C03644=1019.248,-10.777,397.334,166.343,52.857,159.580
C03645=1019.242,-11.026,397.348,166.340,52.863,159.581
C03646=1019.236,-11.276,397.360,166.337,52.868,159.581
C03647=1019.231,-11.525,397.374,166.334,52.874,159.582
C03648=1019.225,-11.775,397.386,166.331,52.880,159.582
C03649=1019.220,-12.024,397.400,166.328,52.885,159.583
C03650=1019.214,-12.274,397.413,166.325,52.891,159.583
C03651=1019.208,-12.523,397.426,166.322,52.896,159.583
C03652=1019.203,-12.773,397.439,166.321,52.902,159.584
C03653=1019.197,-13.023,397.451,166.318,52.907,159.584
C03654=1019.192,-13.272,397.465,166.315,52.913,159.585
C03655=1019.186,-13.522,397.478,166.312,52.919,159.586
C03656=1019.180,-13.771,397.490,166.309,52.924,159.586
C03657=1019.175,-14.021,397.504,166.306,52.929,159.586
C03658=1019.169,-14.271,397.516,166.303,52.935,159.587
C03659=1019.164,-14.521,397.530,166.301,52.941,159.587
C03660=1019.158,-14.770,397.542,166.299,52.946,159.588
C03661=1019.153,-15.020,397.555,166.296,52.951,159.588
C03662=1019.147,-15.269,397.569,166.293,52.957,159.589
C03663=1019.141,-15.519,397.581,166.290,52.962,159.589
C03664=1019.137,-15.769,397.594,166.287,52.968,159.590
C03665=1019.130,-16.018,397.607,166.284,52.974,159.590
C03666=1019.124,-16.268,397.620,166.281,52.979,159.591
C03667=1019.118,-16.518,397.632,166.279,52.985,159.591
C03668=1019.113,-16.767,397.645,166.276,52.991,159.592
C03669=1019.108,-17.016,397.658,166.273,52.996,159.592
C03670=1019.102,-17.266,397.671,166.270,53.002,159.593
C03671=1019.096,-17.515,397.683,166.267,53.007,159.593
C03672=1019.091,-17.765,397.696,166.265,53.014,159.594
C03673=1019.085,-18.015,397.708,166.263,53.019,159.594
C03674=1019.079,-18.265,397.721,166.260,53.024,159.595
C03675=1019.073,-18.514,397.733,166.257,53.030,159.595
C03676=1019.068,-18.764,397.747,166.254,53.035,159.596
C03677=1019.062,-19.014,397.759,166.251,53.041,159.596
C03678=1019.057,-19.263,397.772,166.249,53.047,159.597
C03679=1019.051,-19.513,397.784,166.246,53.052,159.597
C03680=1019.045,-19.763,397.797,166.243,53.058,159.597
C03681=1019.040,-20.012,397.809,166.240,53.064,159.598
C03682=1019.034,-20.262,397.821,166.237,53.069,159.598
C03683=1019.028,-20.512,397.834,166.234,53.075,159.599
C03684=1019.023,-20.761,397.847,166.231,53.080,159.599
C03685=1019.016,-21.039,397.861,166.229,53.086,159.600
C03686=1019.010,-21.317,397.875,166.225,53.093,159.600
C03687=1019.004,-21.596,397.888,166.223,53.099,159.601
C03688=1018.998,-21.874,397.903,166.219,53.105,159.601
C03689=1018.992,-22.124,397.915,166.216,53.111,159.602
C03690=1018.986,-22.374,397.928,166.213,53.117,159.602
C03691=1018.981,-22.623,397.940,166.210,53.122,159.603
C03692=1018.975,-22.873,397.952,166.207,53.128,159.603
C03693=1018.970,-23.122,397.965,166.204,53.133,159.604
C03694=1018.964,-23.372,397.978,166.201,53.139,159.604
C03695=1018.958,-23.622,397.991,166.199,53.145,159.605
C03696=1018.953,-23.872,398.002,166.197,53.150,159.605
C03697=1018.947,-24.122,398.015,166.194,53.155,159.605
C03698=1018.942,-24.371,398.027,166.191,53.161,159.606
C03699=1018.936,-24.621,398.040,166.189,53.167,159.607
C03700=1018.931,-24.870,398.052,166.186,53.172,159.607
C03701=1018.925,-25.120,398.064,166.183,53.177,159.607
C03702=1018.919,-25.370,398.077,166.180,53.183,159.608
C03703=1018.914,-25.619,398.090,166.177,53.188,159.608
C03704=1018.909,-25.869,398.102,166.174,53.194,159.609
C03705=1018.903,-26.118,398.115,166.171,53.200,159.609
C03706=1018.897,-26.368,398.127,166.168,53.205,159.609
C03707=1018.892,-26.617,398.139,166.165,53.211,159.610
C03708=1018.886,-26.867,398.152,166.163,53.216,159.610
C03709=1018.881,-27.116,398.164,166.160,53.221,159.611
C03710=1018.875,-27.366,398.177,166.157,53.227,159.611
C03711=1018.870,-27.616,398.188,166.155,53.233,159.612
C03712=1018.864,-27.866,398.201,166.152,53.238,159.612
C03713=1018.858,-28.116,398.213,166.149,53.244,159.613
C03714=1018.853,-28.365,398.225,166.146,53.250,159.613
C03715=1018.847,-28.615,398.237,166.143,53.255,159.614
C03716=1018.842,-28.865,398.249,166.140,53.261,159.614
C03717=1018.835,-29.114,398.261,166.137,53.266,159.614
C03718=1018.830,-29.363,398.274,166.135,53.272,159.615
C03719=1018.825,-29.613,398.285,166.132,53.278,159.615
C03720=1018.819,-29.863,398.298,166.129,53.283,159.616
C03721=1018.814,-30.112,398.310,166.126,53.289,159.616
C03722=1018.808,-30.363,398.322,166.123,53.295,159.617
C03723=1018.802,-30.612,398.333,166.120,53.300,159.617
C03724=1018.796,-30.862,398.346,166.118,53.306,159.618
C03725=1018.791,-31.111,398.357,166.115,53.312,159.618
C03726=1018.785,-31.361,398.370,166.112,53.317,159.619
C03727=1018.780,-31.610,398.382,166.109,53.322,159.619
C03728=1018.774,-31.861,398.394,166.107,53.329,159.620
C03729=1018.768,-32.110,398.405,166.104,53.334,159.620
C03730=1018.763,-32.359,398.418,166.101,53.339,159.620
C03731=1018.757,-32.609,398.429,166.098,53.345,159.621
C03732=1018.752,-32.859,398.442,166.095,53.350,159.621
C03733=1018.746,-33.109,398.454,166.092,53.356,159.622
C03734=1018.740,-33.358,398.465,166.089,53.362,159.622
C03735=1018.734,-33.608,398.478,166.086,53.367,159.623
C03736=1018.729,-33.858,398.489,166.083,53.373,159.623
C03737=1018.724,-34.107,398.501,166.081,53.379,159.624
C03738=1018.718,-34.357,398.514,166.078,53.384,159.624
C03739=1018.713,-34.606,398.525,166.075,53.390,159.624
C03740=1018.707,-34.855,398.537,166.072,53.395,159.625
C03741=1018.702,-35.106,398.549,166.069,53.401,159.625
C03742=1018.696,-35.355,398.561,166.066,53.406,159.626
C03743=1018.691,-35.606,398.573,166.064,53.412,159.626
C03744=1018.685,-35.855,398.585,166.061,53.418,159.627
C03745=1018.680,-36.104,398.596,166.058,53.423,159.627
C03746=1018.674,-36.354,398.608,166.055,53.429,159.627
C03747=1018.669,-36.604,398.620,166.052,53.434,159.628
C03748=1018.663,-36.853,398.632,166.049,53.440,159.628
C03749=1018.658,-37.081,398.642,166.047,53.445,159.629
C03750=1018.653,-37.308,398.654,166.044,53.450,159.629
C03751=1018.649,-37.536,398.664,166.040,53.455,159.629
C03752=1018.643,-37.764,398.674,166.039,53.460,159.630
C03753=1018.638,-37.991,398.686,166.036,53.465,159.630
C03754=1018.633,-38.219,398.696,166.033,53.470,159.630
C03755=1018.629,-38.447,398.707,166.030,53.475,159.631
C03756=1018.624,-38.675,398.718,166.028,53.480,159.631
C03757=1018.617,-38.925,398.730,166.025,53.486,159.632
C03758=1018.612,-39.174,398.742,166.023,53.491,159.632
C03759=1018.607,-39.424,398.753,166.020,53.497,159.633
C03760=1018.601,-39.674,398.765,166.017,53.502,159.633
C03761=1018.595,-39.923,398.777,166.014,53.507,159.633
C03762=1018.590,-40.173,398.788,166.011,53.514,159.634
C03763=1018.584,-40.423,398.799,166.008,53.519,159.634
C03764=1018.579,-40.673,398.811,166.005,53.525,159.635
C03765=1018.573,-40.922,398.822,166.003,53.531,159.635
C03766=1018.568,-41.172,398.834,166.000,53.536,159.636
C03767=1018.562,-41.422,398.845,165.996,53.542,159.636
C03768=1018.557,-41.672,398.857,165.993,53.547,159.636
C03769=1018.551,-41.921,398.868,165.990,53.553,159.637
C03770=1018.546,-42.170,398.880,165.987,53.559,159.637
C03771=1018.539,-42.421,398.891,165.985,53.565,159.638
C03772=1018.534,-42.670,398.902,165.982,53.570,159.638
C03773=1018.528,-42.919,398.914,165.979,53.575,159.638
C03774=1018.523,-43.169,398.925,165.976,53.582,159.639
C03775=1018.517,-43.419,398.936,165.973,53.587,159.639
C03776=1018.512,-43.669,398.948,165.970,53.593,159.640
C03777=1018.506,-43.919,398.959,165.967,53.598,159.640
C03778=1018.501,-44.168,398.971,165.964,53.604,159.641
C03779=1018.496,-44.418,398.983,165.961,53.609,159.641
C03780=1018.490,-44.667,398.994,165.959,53.615,159.642
C03781=1018.484,-44.918,399.005,165.956,53.621,159.642
C03782=1018.479,-45.167,399.016,165.953,53.626,159.642
C03783=1018.474,-45.417,399.028,165.950,53.632,159.643
C03784=1018.468,-45.666,399.039,165.947,53.637,159.643
C03785=1018.463,-45.915,399.051,165.944,53.643,159.644
C03786=1018.457,-46.165,399.062,165.941,53.648,159.644
C03787=1018.451,-46.415,399.074,165.939,53.654,159.645
C03788=1018.446,-46.665,399.084,165.936,53.660,159.645
C03789=1018.441,-46.915,399.096,165.933,53.665,159.645
C03790=1018.435,-47.164,399.107,165.930,53.671,159.646
C03791=1018.430,-47.414,399.118,165.927,53.676,159.646
C03792=1018.424,-47.664,399.129,165.924,53.682,159.646
C03793=1018.419,-47.913,399.141,165.921,53.687,159.647
C03794=1018.413,-48.163,399.151,165.918,53.692,159.647
C03795=1018.408,-48.413,399.163,165.915,53.698,159.648
C03796=1018.402,-48.662,399.175,165.913,53.703,159.648
C03797=1018.397,-48.912,399.186,165.910,53.710,159.649
C03798=1018.391,-49.161,399.197,165.907,53.715,159.649
C03799=1018.386,-49.411,399.209,165.904,53.721,159.649
C03800=1018.380,-49.661,399.220,165.901,53.726,159.650
C03801=1018.375,-49.911,399.231,165.898,53.732,159.650
C03802=1018.369,-50.160,399.242,165.895,53.737,159.650
C03803=1018.364,-50.410,399.253,165.892,53.743,159.651
C03804=1018.359,-50.659,399.264,165.890,53.748,159.651
C03805=1018.354,-50.909,399.276,165.887,53.753,159.652
C03806=1018.348,-51.159,399.286,165.883,53.759,159.652
C03807=1018.342,-51.409,399.297,165.880,53.765,159.652
C03808=1018.336,-51.659,399.308,165.877,53.771,159.653
C03809=1018.330,-51.981,399.322,165.874,53.778,159.654
C03810=1018.322,-52.302,399.336,165.870,53.785,159.654
C03811=1018.315,-52.623,399.349,165.866,53.793,159.654
C03812=1018.308,-52.944,399.364,165.863,53.800,159.655
C03813=1018.302,-53.222,399.375,165.859,53.807,159.656
C03814=1018.295,-53.500,399.387,165.856,53.813,159.656
C03815=1018.289,-53.778,399.400,165.852,53.820,159.656
C03816=1018.283,-54.056,399.411,165.850,53.826,159.657
C03817=1018.277,-54.306,399.422,165.847,53.832,159.657
C03818=1018.272,-54.555,399.433,165.843,53.838,159.658
C03819=1018.266,-54.805,399.443,165.840,53.843,159.658
C03820=1018.260,-55.055,399.454,165.837,53.849,159.659
C03821=1018.255,-55.304,399.465,165.834,53.855,159.659
C03822=1018.249,-55.554,399.475,165.831,53.860,159.659
C03823=1018.243,-55.804,399.486,165.829,53.866,159.660
C03824=1018.238,-56.054,399.497,165.826,53.872,159.660
C03825=1018.233,-56.304,399.508,165.822,53.878,159.661
C03826=1018.227,-56.553,399.519,165.819,53.883,159.661
C03827=1018.222,-56.803,399.529,165.816,53.889,159.661
C03828=1018.217,-57.052,399.539,165.813,53.894,159.662
C03829=1018.211,-57.302,399.550,165.811,53.901,159.662
C03830=1018.206,-57.552,399.560,165.808,53.906,159.663
C03831=1018.200,-57.801,399.571,165.805,53.912,159.663
C03832=1018.194,-58.051,399.582,165.801,53.917,159.663
C03833=1018.189,-58.301,399.592,165.798,53.923,159.664
C03834=1018.183,-58.550,399.603,165.796,53.929,159.664
C03835=1018.177,-58.800,399.613,165.793,53.935,159.665
C03836=1018.172,-59.050,399.625,165.790,53.940,159.665
C03837=1018.167,-59.300,399.636,165.787,53.946,159.665
C03838=1018.161,-59.550,399.646,165.784,53.951,159.666
C03839=1018.156,-59.799,399.656,165.781,53.957,159.666
C03840=1018.151,-60.049,399.666,165.779,53.963,159.667
C03841=1018.145,-60.298,399.677,165.775,53.969,159.667
C03842=1018.140,-60.548,399.687,165.772,53.974,159.667
C03843=1018.134,-60.798,399.698,165.769,53.980,159.668
C03844=1018.128,-61.048,399.708,165.766,53.985,159.668
C03845=1018.123,-61.297,399.719,165.763,53.991,159.669
C03846=1018.118,-61.547,399.729,165.760,53.996,159.669
C03847=1018.112,-61.796,399.740,165.757,54.002,159.669
C03848=1018.107,-62.046,399.750,165.755,54.007,159.670
C03849=1018.102,-62.296,399.762,165.752,54.014,159.670
C03850=1018.096,-62.546,399.772,165.749,54.019,159.671
C03851=1018.090,-62.796,399.783,165.745,54.025,159.671
C03852=1018.086,-63.045,399.792,165.742,54.031,159.671
C03853=1018.080,-63.295,399.803,165.739,54.036,159.672
C03854=1018.074,-63.545,399.813,165.737,54.042,159.672
C03855=1018.069,-63.795,399.824,165.734,54.047,159.672
C03856=1018.064,-64.044,399.834,165.731,54.053,159.673
C03857=1018.058,-64.294,399.844,165.728,54.058,159.673
C03858=1018.053,-64.544,399.854,165.725,54.064,159.673
C03859=1018.047,-64.793,399.865,165.722,54.069,159.674
C03860=1018.042,-65.044,399.876,165.719,54.075,159.674
C03861=1018.037,-65.292,399.886,165.716,54.080,159.675
C03862=1018.031,-65.542,399.896,165.713,54.086,159.675
C03863=1018.026,-65.793,399.906,165.709,54.092,159.675
C03864=1018.020,-66.042,399.917,165.707,54.097,159.676
C03865=1018.015,-66.291,399.927,165.704,54.103,159.676
C03866=1018.011,-66.542,399.938,165.701,54.108,159.676
C03867=1018.005,-66.791,399.949,165.698,54.114,159.677
C03868=1018.000,-67.041,399.958,165.695,54.119,159.677
C03869=1017.995,-67.291,399.969,165.692,54.125,159.677
C03870=1017.989,-67.540,399.980,165.689,54.130,159.678
C03871=1017.983,-67.791,399.990,165.686,54.136,159.678
C03872=1017.979,-68.040,399.999,165.683,54.141,159.678
C03873=1017.973,-68.289,400.010,165.680,54.147,159.679
C03874=1017.967,-68.540,400.020,165.678,54.152,159.679
C03875=1017.963,-68.789,400.030,165.675,54.158,159.680
C03876=1017.957,-69.039,400.040,165.672,54.163,159.680
C03877=1017.951,-69.318,400.052,165.668,54.170,159.680
C03878=1017.945,-69.597,400.064,165.665,54.176,159.681
C03879=1017.940,-69.876,400.075,165.662,54.182,159.681
C03880=1017.933,-70.155,400.086,165.658,54.188,159.681
C03881=1017.928,-70.405,400.096,165.655,54.194,159.682
C03882=1017.923,-70.654,400.107,165.652,54.199,159.682
C03883=1017.917,-70.904,400.117,165.649,54.205,159.683
C03884=1017.912,-71.154,400.127,165.647,54.210,159.683
C03885=1017.907,-71.403,400.137,165.644,54.216,159.683
C03886=1017.902,-71.653,400.147,165.640,54.221,159.683
C03887=1017.897,-71.902,400.158,165.637,54.226,159.684
C03888=1017.891,-72.152,400.168,165.634,54.232,159.684
C03889=1017.886,-72.402,400.178,165.632,54.237,159.685
C03890=1017.881,-72.652,400.188,165.629,54.243,159.685
C03891=1017.875,-72.902,400.198,165.626,54.248,159.685
C03892=1017.871,-73.151,400.208,165.623,54.254,159.686
C03893=1017.865,-73.401,400.218,165.620,54.259,159.686
C03894=1017.860,-73.651,400.229,165.617,54.264,159.686
C03895=1017.855,-73.901,400.239,165.614,54.270,159.686
C03896=1017.850,-74.151,400.249,165.611,54.275,159.687
C03897=1017.845,-74.400,400.259,165.608,54.281,159.687
C03898=1017.839,-74.650,400.269,165.605,54.286,159.688
C03899=1017.834,-74.899,400.279,165.602,54.292,159.688
C03900=1017.829,-75.149,400.289,165.599,54.297,159.688
C03901=1017.823,-75.399,400.299,165.597,54.303,159.689
C03902=1017.818,-75.649,400.308,165.593,54.309,159.689
C03903=1017.812,-75.899,400.318,165.590,54.314,159.689
C03904=1017.808,-76.149,400.327,165.587,54.320,159.690
C03905=1017.802,-76.399,400.337,165.584,54.325,159.690
C03906=1017.797,-76.648,400.347,165.581,54.331,159.690
C03907=1017.791,-76.898,400.357,165.578,54.337,159.691
C03908=1017.786,-77.147,400.367,165.575,54.342,159.691
C03909=1017.780,-77.397,400.376,165.573,54.348,159.691
C03910=1017.775,-77.647,400.386,165.569,54.354,159.692
C03911=1017.770,-77.897,400.396,165.566,54.359,159.692
C03912=1017.765,-78.147,400.405,165.563,54.365,159.692
C03913=1017.759,-78.397,400.415,165.560,54.370,159.693
C03914=1017.754,-78.646,400.425,165.557,54.376,159.693
C03915=1017.749,-78.896,400.435,165.554,54.381,159.693
C03916=1017.744,-79.146,400.445,165.551,54.387,159.694
C03917=1017.739,-79.395,400.454,165.548,54.392,159.694
C03918=1017.734,-79.645,400.463,165.546,54.398,159.695
C03919=1017.729,-79.895,400.473,165.543,54.404,159.695
C03920=1017.722,-80.145,400.483,165.539,54.409,159.695
C03921=1017.718,-80.394,400.492,165.536,54.415,159.696
C03922=1017.712,-80.644,400.501,165.533,54.421,159.696
C03923=1017.707,-80.894,400.511,165.530,54.426,159.696
C03924=1017.701,-81.144,400.521,165.527,54.432,159.697
C03925=1017.696,-81.394,400.530,165.524,54.437,159.697
C03926=1017.691,-81.643,400.539,165.521,54.444,159.697
C03927=1017.685,-81.893,400.549,165.518,54.450,159.698
C03928=1017.680,-82.143,400.557,165.515,54.455,159.698
C03929=1017.675,-82.393,400.568,165.512,54.461,159.698
C03930=1017.669,-82.642,400.576,165.510,54.466,159.699
C03931=1017.664,-82.891,400.585,165.506,54.472,159.699
C03932=1017.658,-83.142,400.595,165.503,54.478,159.699
C03933=1017.653,-83.391,400.604,165.500,54.483,159.700
C03934=1017.648,-83.641,400.614,165.497,54.489,159.700
C03935=1017.642,-83.891,400.623,165.495,54.495,159.701
C03936=1017.638,-84.140,400.632,165.491,54.501,159.701
C03937=1017.632,-84.391,400.641,165.488,54.507,159.701
C03938=1017.627,-84.640,400.651,165.485,54.512,159.702
C03939=1017.622,-84.890,400.660,165.482,54.518,159.702
C03940=1017.615,-85.140,400.669,165.479,54.523,159.702
C03941=1017.610,-85.421,400.680,165.476,54.530,159.703
C03942=1017.604,-85.701,400.690,165.472,54.536,159.703
C03943=1017.598,-85.983,400.701,165.469,54.543,159.703
C03944=1017.592,-86.263,400.711,165.466,54.549,159.704
C03945=1017.587,-86.513,400.720,165.462,54.555,159.704
C03946=1017.582,-86.762,400.729,165.459,54.561,159.705
C03947=1017.577,-87.013,400.738,165.457,54.566,159.705
C03948=1017.571,-87.262,400.748,165.454,54.572,159.705
C03949=1017.566,-87.512,400.756,165.451,54.577,159.706
C03950=1017.560,-87.762,400.766,165.448,54.583,159.706
C03951=1017.555,-88.012,400.775,165.445,54.588,159.706
C03952=1017.551,-88.262,400.784,165.441,54.594,159.707
C03953=1017.545,-88.511,400.793,165.438,54.600,159.707
C03954=1017.540,-88.762,400.802,165.436,54.605,159.707
C03955=1017.534,-89.011,400.812,165.433,54.611,159.708
C03956=1017.529,-89.260,400.820,165.430,54.617,159.708
C03957=1017.524,-89.510,400.829,165.427,54.622,159.708
C03958=1017.518,-89.760,400.839,165.424,54.627,159.708
C03959=1017.514,-90.010,400.848,165.420,54.633,159.709
C03960=1017.508,-90.260,400.856,165.417,54.639,159.709
C03961=1017.503,-90.509,400.866,165.414,54.644,159.709
C03962=1017.498,-90.759,400.875,165.411,54.650,159.710
C03963=1017.492,-91.009,400.884,165.408,54.655,159.710
C03964=1017.488,-91.259,400.893,165.406,54.661,159.710
C03965=1017.482,-91.509,400.902,165.403,54.667,159.711
C03966=1017.478,-91.759,400.911,165.400,54.672,159.711
C03967=1017.472,-92.008,400.920,165.397,54.678,159.712
C03968=1017.466,-92.258,400.929,165.393,54.684,159.712
C03969=1017.462,-92.508,400.938,165.390,54.689,159.712
C03970=1017.456,-92.757,400.947,165.387,54.695,159.712
C03971=1017.452,-93.007,400.956,165.384,54.700,159.713
C03972=1017.447,-93.257,400.965,165.381,54.705,159.713
C03973=1017.441,-93.507,400.973,165.378,54.711,159.713
C03974=1017.436,-93.756,400.983,165.376,54.716,159.714
C03975=1017.431,-94.007,400.992,165.373,54.722,159.714
C03976=1017.426,-94.257,401.001,165.370,54.728,159.714
C03977=1017.421,-94.506,401.009,165.367,54.733,159.715
C03978=1017.415,-94.755,401.019,165.364,54.739,159.715
C03979=1017.411,-95.006,401.028,165.361,54.744,159.715
C03980=1017.405,-95.255,401.036,165.357,54.750,159.715
C03981=1017.401,-95.505,401.045,165.354,54.755,159.716
C03982=1017.395,-95.754,401.054,165.351,54.761,159.716
C03983=1017.390,-96.004,401.063,165.348,54.766,159.716
C03984=1017.385,-96.255,401.072,165.345,54.771,159.717
C03985=1017.380,-96.505,401.081,165.342,54.777,159.717
C03986=1017.375,-96.755,401.090,165.339,54.783,159.717
C03987=1017.370,-97.004,401.098,165.337,54.788,159.718
C03988=1017.364,-97.253,401.108,165.334,54.794,159.718
C03989=1017.360,-97.503,401.117,165.330,54.799,159.718
///RCONF 1,0,0,0,1,0,0,0,0,0,0,0,0,0,0,0,0,0,0,0,0,0,0,0
C03990=1017.355,-97.753,401.125,165.328,54.804,159.718
C03991=1017.349,-98.003,401.134,165.325,54.810,159.719
C03992=1017.345,-98.253,401.143,165.322,54.815,159.719
C03993=1017.340,-98.503,401.151,165.319,54.821,159.719
C03994=1017.334,-98.752,401.160,165.315,54.827,159.720
C03995=1017.329,-99.002,401.168,165.312,54.833,159.720
C03996=1017.324,-99.252,401.177,165.310,54.838,159.720
C03997=1017.318,-99.501,401.185,165.307,54.844,159.721
C03998=1017.313,-99.751,401.194,165.304,54.849,159.721
C03999=1017.308,-100.001,401.201,165.301,54.855,159.721
C04000=1017.303,-100.251,401.210,165.297,54.861,159.722
C04001=1017.298,-100.501,401.219,165.294,54.867,159.722
C04002=1017.293,-100.751,401.228,165.292,54.872,159.722
C04003=1017.288,-101.001,401.236,165.289,54.878,159.723
C04004=1017.283,-101.250,401.244,165.286,54.883,159.723
C04005=1017.277,-101.534,401.254,165.282,54.889,159.723
C04006=1017.271,-101.816,401.263,165.279,54.896,159.724
C04007=1017.265,-102.100,401.273,165.275,54.902,159.724
C04008=1017.259,-102.383,401.283,165.272,54.908,159.724
C04009=1017.254,-102.632,401.291,165.270,54.914,159.725
C04010=1017.249,-102.882,401.300,165.266,54.920,159.725
C04011=1017.243,-103.132,401.308,165.263,54.926,159.725
C04012=1017.238,-103.382,401.317,165.260,54.931,159.726
C04013=1017.233,-103.632,401.324,165.257,54.937,159.726
C04014=1017.229,-103.882,401.333,165.254,54.942,159.726
C04015=1017.224,-104.131,401.342,165.251,54.947,159.726
C04016=1017.219,-104.381,401.350,165.248,54.953,159.727
C04017=1017.214,-104.630,401.359,165.245,54.959,159.727
C04018=1017.209,-104.881,401.366,165.243,54.964,159.727
C04019=1017.203,-105.130,401.375,165.239,54.970,159.728
C04020=1017.198,-105.380,401.383,165.236,54.976,159.728
C04021=1017.193,-105.630,401.392,165.233,54.982,159.728
C04022=1017.188,-105.880,401.400,165.230,54.986,159.728
C04023=1017.183,-106.130,401.408,165.227,54.992,159.729
C04024=1017.178,-106.379,401.416,165.224,54.998,159.729
C04025=1017.173,-106.629,401.425,165.221,55.003,159.729
C04026=1017.168,-106.879,401.432,165.218,55.009,159.730
C04027=1017.162,-107.129,401.441,165.216,55.015,159.730
C04028=1017.157,-107.378,401.449,165.213,55.020,159.731
C04029=1017.152,-107.629,401.457,165.209,55.026,159.731
C04030=1017.148,-107.878,401.465,165.206,55.031,159.731
C04031=1017.142,-108.127,401.474,165.203,55.037,159.731
C04032=1017.137,-108.378,401.482,165.200,55.042,159.731
C04033=1017.132,-108.628,401.490,165.197,55.048,159.732
C04034=1017.127,-108.878,401.498,165.194,55.054,159.732
C04035=1017.122,-109.128,401.506,165.192,55.059,159.733
C04036=1017.117,-109.377,401.514,165.188,55.065,159.733
C04037=1017.112,-109.627,401.522,165.185,55.071,159.733
C04038=1017.107,-109.877,401.530,165.182,55.076,159.733
C04039=1017.101,-110.127,401.538,165.179,55.082,159.734
C04040=1017.096,-110.376,401.546,165.176,55.088,159.734
C04041=1017.092,-110.626,401.554,165.174,55.093,159.734
C04042=1017.086,-110.876,401.562,165.170,55.098,159.735
C04043=1017.081,-111.126,401.570,165.168,55.104,159.735
C04044=1017.076,-111.376,401.578,165.165,55.110,159.735
C04045=1017.072,-111.625,401.586,165.161,55.116,159.735
C04046=1017.066,-111.875,401.594,165.158,55.121,159.736
C04047=1017.062,-112.125,401.602,165.155,55.127,159.736
C04048=1017.056,-112.375,401.609,165.152,55.132,159.736
C04049=1017.051,-112.625,401.617,165.149,55.137,159.736
C04050=1017.046,-112.875,401.625,165.146,55.143,159.737
C04051=1017.041,-113.125,401.634,165.144,55.149,159.737
C04052=1017.037,-113.374,401.641,165.141,55.154,159.738
C04053=1017.031,-113.624,401.650,165.138,55.160,159.738
C04054=1017.026,-113.874,401.657,165.135,55.166,159.738
C04055=1017.022,-114.123,401.665,165.132,55.170,159.738
C04056=1017.016,-114.373,401.673,165.128,55.176,159.738
C04057=1017.011,-114.624,401.680,165.125,55.182,159.739
C04058=1017.006,-114.873,401.689,165.122,55.188,159.739
C04059=1017.001,-115.123,401.696,165.120,55.193,159.740
C04060=1016.996,-115.373,401.704,165.117,55.199,159.740
C04061=1016.991,-115.622,401.712,165.114,55.205,159.740
C04062=1016.986,-115.872,401.719,165.111,55.210,159.741
C04063=1016.981,-116.123,401.727,165.108,55.215,159.741
C04064=1016.976,-116.372,401.735,165.105,55.221,159.741
C04065=1016.971,-116.622,401.742,165.102,55.227,159.741
C04066=1016.966,-116.872,401.750,165.098,55.233,159.741
C04067=1016.961,-117.122,401.758,165.096,55.238,159.742
C04068=1016.956,-117.371,401.766,165.093,55.244,159.742
C04069=1016.950,-117.655,401.774,165.089,55.250,159.742
C04070=1016.945,-117.938,401.782,165.087,55.256,159.743
C04071=1016.939,-118.220,401.792,165.083,55.262,159.743
C04072=1016.933,-118.504,401.800,165.079,55.269,159.743
C04073=1016.929,-118.754,401.808,165.077,55.275,159.744
C04074=1016.923,-119.003,401.815,165.073,55.280,159.744
C04075=1016.918,-119.254,401.823,165.071,55.285,159.744
C04076=1016.914,-119.503,401.831,165.068,55.291,159.745
C04077=1016.908,-119.753,401.838,165.065,55.297,159.745
C04078=1016.904,-120.002,401.845,165.062,55.302,159.745
C04079=1016.899,-120.253,401.853,165.059,55.308,159.746
C04080=1016.893,-120.503,401.860,165.056,55.313,159.746
C04081=1016.889,-120.752,401.868,165.052,55.319,159.746
C04082=1016.884,-121.003,401.875,165.049,55.325,159.746
C04083=1016.879,-121.252,401.884,165.047,55.330,159.747
C04084=1016.873,-121.502,401.891,165.044,55.336,159.747
C04085=1016.869,-121.751,401.898,165.041,55.341,159.747
C04086=1016.864,-122.002,401.906,165.038,55.346,159.747
C04087=1016.859,-122.251,401.913,165.035,55.352,159.748
C04088=1016.854,-122.501,401.920,165.032,55.358,159.748
C04089=1016.849,-122.751,401.927,165.029,55.363,159.748
C04090=1016.844,-123.001,401.935,165.027,55.369,159.749
C04091=1016.840,-123.251,401.942,165.023,55.374,159.749
C04092=1016.834,-123.501,401.950,165.021,55.380,159.749
C04093=1016.830,-123.750,401.957,165.018,55.385,159.749
C04094=1016.825,-124.001,401.965,165.015,55.391,159.750
C04095=1016.820,-124.250,401.972,165.012,55.396,159.750
C04096=1016.815,-124.500,401.979,165.009,55.402,159.750
C04097=1016.810,-124.750,401.987,165.006,55.407,159.751
C04098=1016.805,-125.000,401.994,165.003,55.413,159.751
C04099=1016.800,-125.249,402.001,164.999,55.419,159.751
C04100=1016.795,-125.499,402.008,164.997,55.425,159.751
C04101=1016.790,-125.749,402.016,164.993,55.430,159.751
C04102=1016.785,-125.998,402.023,164.991,55.435,159.752
C04103=1016.780,-126.249,402.030,164.988,55.441,159.752
C04104=1016.775,-126.499,402.037,164.985,55.447,159.752
C04105=1016.770,-126.749,402.044,164.982,55.452,159.753
C04106=1016.765,-126.998,402.051,164.979,55.457,159.753
C04107=1016.761,-127.248,402.059,164.976,55.463,159.753
C04108=1016.755,-127.498,402.066,164.973,55.469,159.754
C04109=1016.751,-127.748,402.073,164.971,55.474,159.754
C04110=1016.746,-127.997,402.080,164.968,55.480,159.754
C04111=1016.741,-128.247,402.087,164.965,55.485,159.754
C04112=1016.737,-128.496,402.095,164.961,55.490,159.754
C04113=1016.733,-128.746,402.103,164.959,55.494,159.755
C04114=1016.729,-128.996,402.113,164.956,55.498,159.755
C04115=1016.726,-129.246,402.122,164.953,55.501,159.754
C04116=1016.723,-129.495,402.132,164.951,55.504,159.754
C04117=1016.721,-129.744,402.144,164.948,55.506,159.754
C04118=1016.719,-129.994,402.155,164.946,55.507,159.754
C04119=1016.717,-130.244,402.167,164.943,55.508,159.753
C04120=1016.716,-130.493,402.179,164.941,55.509,159.753
C04121=1016.716,-130.743,402.193,164.939,55.507,159.752
C04122=1016.715,-130.993,402.206,164.937,55.507,159.752
C04123=1016.715,-131.242,402.221,164.935,55.505,159.751
C04124=1016.715,-131.492,402.236,164.932,55.503,159.750
C04125=1016.716,-131.742,402.252,164.930,55.501,159.749
C04126=1016.717,-131.991,402.268,164.928,55.498,159.748
C04127=1016.719,-132.241,402.285,164.926,55.495,159.747
C04128=1016.720,-132.491,402.302,164.924,55.490,159.746
C04129=1016.723,-132.741,402.320,164.922,55.486,159.744
C04130=1016.726,-132.991,402.339,164.921,55.480,159.743
C04131=1016.728,-133.240,402.358,164.920,55.474,159.742
C04132=1016.733,-133.489,402.378,164.918,55.468,159.740
C04133=1016.478,-133.516,401.988,164.879,55.831,159.794
C04134=1016.475,-133.267,401.968,164.880,55.837,159.796
C04135=1016.471,-133.017,401.949,164.882,55.843,159.797
C04136=1016.469,-132.767,401.930,164.884,55.848,159.799
C04137=1016.466,-132.517,401.912,164.886,55.852,159.800
C04138=1016.464,-132.268,401.894,164.888,55.857,159.801
C04139=1016.463,-132.018,401.877,164.889,55.860,159.802
C04140=1016.462,-131.768,401.862,164.891,55.863,159.803
C04141=1016.461,-131.518,401.846,164.893,55.866,159.804
C04142=1016.460,-131.268,401.831,164.896,55.868,159.805
C04143=1016.461,-131.019,401.817,164.898,55.869,159.806
C04144=1016.461,-130.769,401.803,164.900,55.870,159.807
C04145=1016.462,-130.519,401.790,164.903,55.870,159.807
C04146=1016.463,-130.270,401.777,164.905,55.870,159.808
C04147=1016.464,-130.020,401.765,164.908,55.870,159.808
C04148=1016.466,-129.771,401.753,164.909,55.868,159.809
C04149=1016.469,-129.521,401.743,164.912,55.866,159.809
C04150=1016.472,-129.272,401.732,164.915,55.863,159.809
C04151=1016.474,-129.022,401.722,164.917,55.860,159.809
C04152=1016.478,-128.772,401.714,164.920,55.856,159.809
C04153=1016.482,-128.523,401.705,164.922,55.852,159.809
C04154=1016.487,-128.273,401.697,164.925,55.847,159.809
C04155=1016.491,-128.023,401.690,164.929,55.842,159.809
C04156=1016.496,-127.774,401.683,164.931,55.836,159.808
C04157=1016.501,-127.524,401.676,164.934,55.831,159.808
C04158=1016.506,-127.275,401.669,164.937,55.825,159.808
C04159=1016.511,-127.024,401.661,164.940,55.819,159.807
C04160=1016.516,-126.775,401.654,164.943,55.813,159.807
C04161=1016.520,-126.525,401.647,164.947,55.808,159.807
C04162=1016.525,-126.275,401.640,164.949,55.802,159.807
C04163=1016.530,-126.025,401.633,164.952,55.797,159.806
C04164=1016.536,-125.775,401.626,164.955,55.791,159.806
C04165=1016.540,-125.526,401.618,164.958,55.785,159.806
C04166=1016.545,-125.276,401.612,164.960,55.780,159.805
C04167=1016.550,-125.026,401.604,164.963,55.774,159.805
C04168=1016.555,-124.777,401.597,164.967,55.768,159.805
C04169=1016.560,-124.526,401.589,164.970,55.762,159.805
C04170=1016.564,-124.276,401.583,164.973,55.757,159.804
C04171=1016.570,-124.026,401.575,164.976,55.751,159.804
C04172=1016.574,-123.776,401.568,164.978,55.746,159.804
C04173=1016.578,-123.527,401.561,164.981,55.740,159.803
C04174=1016.584,-123.277,401.553,164.984,55.734,159.803
C04175=1016.589,-123.027,401.546,164.986,55.729,159.803
C04176=1016.594,-122.777,401.539,164.990,55.724,159.803
C04177=1016.599,-122.527,401.531,164.992,55.718,159.802
C04178=1016.604,-122.277,401.524,164.996,55.712,159.802
C04179=1016.609,-122.028,401.516,164.999,55.706,159.802
C04180=1016.614,-121.778,401.508,165.002,55.700,159.801
C04181=1016.618,-121.528,401.501,165.005,55.695,159.801
C04182=1016.624,-121.278,401.494,165.007,55.689,159.801
C04183=1016.628,-121.029,401.486,165.010,55.683,159.800
C04184=1016.633,-120.778,401.479,165.013,55.678,159.800
C04185=1016.638,-120.529,401.472,165.016,55.673,159.800
C04186=1016.643,-120.279,401.464,165.020,55.667,159.800
C04187=1016.648,-120.029,401.457,165.023,55.661,159.800
C04188=1016.653,-119.779,401.449,165.025,55.655,159.799
C04189=1016.658,-119.529,401.442,165.028,55.650,159.799
C04190=1016.663,-119.279,401.434,165.031,55.644,159.798
C04191=1016.667,-119.030,401.426,165.034,55.638,159.798
C04192=1016.673,-118.780,401.419,165.036,55.633,159.798
C04193=1016.677,-118.530,401.412,165.040,55.626,159.798
C04194=1016.683,-118.247,401.403,165.043,55.621,159.797
C04195=1016.689,-117.965,401.394,165.046,55.614,159.797
C04196=1016.694,-117.681,401.386,165.050,55.608,159.797
C04197=1016.700,-117.398,401.377,165.053,55.601,159.796
C04198=1016.705,-117.148,401.370,165.056,55.595,159.796
C04199=1016.710,-116.899,401.362,165.059,55.590,159.796
C04200=1016.715,-116.649,401.354,165.062,55.584,159.795
C04201=1016.720,-116.399,401.347,165.065,55.579,159.795
C04202=1016.725,-116.149,401.339,165.069,55.573,159.795
C04203=1016.730,-115.899,401.331,165.071,55.567,159.795
C04204=1016.735,-115.650,401.324,165.074,55.562,159.794
C04205=1016.740,-115.399,401.316,165.077,55.556,159.794
C04206=1016.745,-115.150,401.308,165.080,55.550,159.794
C04207=1016.750,-114.900,401.300,165.082,55.545,159.793
C04208=1016.755,-114.650,401.293,165.086,55.539,159.793
C04209=1016.760,-114.400,401.286,165.089,55.533,159.793
C04210=1016.765,-114.151,401.277,165.092,55.527,159.792
C04211=1016.770,-113.900,401.269,165.094,55.522,159.792
C04212=1016.775,-113.651,401.261,165.097,55.516,159.792
C04213=1016.780,-113.401,401.254,165.100,55.510,159.791
C04214=1016.785,-113.151,401.246,165.103,55.504,159.791
C04215=1016.789,-112.902,401.238,165.107,55.499,159.791
C04216=1016.795,-112.652,401.230,165.110,55.493,159.791
C04217=1016.800,-112.402,401.222,165.113,55.488,159.790
C04218=1016.805,-112.152,401.214,165.115,55.482,159.790
C04219=1016.810,-111.902,401.207,165.118,55.476,159.790
C04220=1016.815,-111.652,401.198,165.121,55.471,159.789
C04221=1016.820,-111.402,401.191,165.125,55.465,159.789
C04222=1016.824,-111.153,401.182,165.127,55.459,159.789
C04223=1016.829,-110.903,401.175,165.130,55.453,159.788
C04224=1016.835,-110.653,401.166,165.133,55.448,159.788
C04225=1016.840,-110.403,401.159,165.136,55.442,159.788
C04226=1016.845,-110.154,401.151,165.140,55.436,159.788
C04227=1016.850,-109.904,401.143,165.142,55.430,159.787
C04228=1016.855,-109.654,401.135,165.145,55.425,159.787
C04229=1016.860,-109.403,401.127,165.148,55.419,159.786
C04230=1016.865,-109.154,401.119,165.151,55.413,159.786
C04231=1016.870,-108.904,401.111,165.154,55.407,159.786
C04232=1016.875,-108.654,401.103,165.157,55.402,159.786
C04233=1016.880,-108.404,401.095,165.160,55.396,159.785
C04234=1016.885,-108.155,401.087,165.163,55.390,159.785
C04235=1016.890,-107.905,401.079,165.166,55.385,159.785
C04236=1016.896,-107.655,401.071,165.169,55.379,159.784
C04237=1016.901,-107.406,401.062,165.172,55.373,159.784
C04238=1016.906,-107.155,401.055,165.175,55.367,159.784
C04239=1016.911,-106.906,401.046,165.178,55.362,159.783
C04240=1016.916,-106.657,401.038,165.180,55.356,159.783
C04241=1016.921,-106.406,401.030,165.183,55.350,159.783
C04242=1016.925,-106.156,401.021,165.187,55.344,159.782
C04243=1016.931,-105.906,401.013,165.190,55.339,159.782
C04244=1016.935,-105.656,401.005,165.193,55.333,159.782
C04245=1016.941,-105.406,400.997,165.195,55.327,159.781
C04246=1016.945,-105.157,400.988,165.199,55.322,159.781
C04247=1016.950,-104.907,400.981,165.201,55.317,159.781
C04248=1016.956,-104.657,400.972,165.205,55.311,159.781
C04249=1016.961,-104.408,400.964,165.208,55.305,159.780
C04250=1016.966,-104.158,400.955,165.211,55.299,159.780
C04251=1016.971,-103.908,400.947,165.214,55.294,159.780
C04252=1016.976,-103.658,400.939,165.216,55.288,159.779
C04253=1016.981,-103.409,400.931,165.219,55.282,159.779
C04254=1016.986,-103.159,400.922,165.223,55.276,159.779
C04255=1016.991,-102.909,400.913,165.226,55.271,159.778
C04256=1016.996,-102.659,400.905,165.229,55.265,159.778
C04257=1017.001,-102.409,400.897,165.231,55.259,159.778
C04258=1017.007,-102.127,400.888,165.235,55.253,159.777
C04259=1017.013,-101.843,400.878,165.238,55.246,159.777
C04260=1017.018,-101.560,400.869,165.242,55.240,159.777
C04261=1017.024,-101.278,400.858,165.245,55.233,159.776
C04262=1017.029,-101.028,400.851,165.248,55.227,159.776
C04263=1017.034,-100.778,400.842,165.251,55.222,159.776
C04264=1017.040,-100.528,400.834,165.254,55.216,159.775
C04265=1017.045,-100.279,400.825,165.257,55.210,159.775
C04266=1017.050,-100.029,400.817,165.260,55.205,159.775
C04267=1017.055,-99.779,400.808,165.263,55.199,159.774
C04268=1017.061,-99.529,400.800,165.266,55.193,159.774
C04269=1017.066,-99.280,400.791,165.269,55.188,159.774
C04270=1017.070,-99.030,400.782,165.272,55.182,159.773
C04271=1017.075,-98.779,400.774,165.275,55.176,159.773
C04272=1017.081,-98.530,400.766,165.277,55.170,159.772
C04273=1017.086,-98.280,400.757,165.280,55.164,159.772
C04274=1017.091,-98.030,400.749,165.284,55.158,159.772
C04275=1017.097,-97.780,400.740,165.287,55.152,159.772
C04276=1017.101,-97.530,400.731,165.290,55.147,159.771
C04277=1017.106,-97.281,400.723,165.293,55.142,159.771
C04278=1017.112,-97.032,400.714,165.296,55.136,159.771
C04279=1017.116,-96.782,400.705,165.299,55.130,159.770
C04280=1017.122,-96.532,400.696,165.301,55.125,159.770
C04281=1017.126,-96.282,400.687,165.305,55.119,159.770
C04282=1017.131,-96.032,400.679,165.308,55.113,159.769
C04283=1017.137,-95.782,400.670,165.311,55.108,159.769
///RCONF 1,0,0,0,0,0,0,0,0,0,0,0,0,0,0,0,0,0,0,0,0,0,0,0
C04284=1017.141,-95.532,400.661,165.314,55.102,159.769
C04285=1017.146,-95.283,400.653,165.316,55.096,159.768
C04286=1017.152,-95.033,400.642,165.319,55.091,159.768
C04287=1017.157,-94.783,400.634,165.322,55.085,159.768
C04288=1017.162,-94.533,400.625,165.326,55.079,159.767
C04289=1017.167,-94.283,400.616,165.329,55.073,159.767
C04290=1017.172,-94.033,400.608,165.332,55.069,159.767
C04291=1017.177,-93.784,400.598,165.335,55.063,159.767
C04292=1017.182,-93.534,400.590,165.338,55.057,159.766
C04293=1017.188,-93.285,400.581,165.340,55.052,159.766
C04294=1017.192,-93.035,400.572,165.344,55.046,159.766
C04295=1017.197,-92.785,400.563,165.347,55.040,159.765
C04296=1017.203,-92.535,400.553,165.350,55.034,159.765
C04297=1017.208,-92.285,400.545,165.353,55.029,159.765
C04298=1017.213,-92.035,400.536,165.355,55.023,159.764
C04299=1017.218,-91.786,400.527,165.358,55.018,159.764
C04300=1017.223,-91.536,400.518,165.362,55.012,159.764
C04301=1017.228,-91.286,400.509,165.365,55.006,159.763
C04302=1017.233,-91.036,400.501,165.368,55.000,159.763
C04303=1017.239,-90.787,400.491,165.370,54.995,159.763
C04304=1017.244,-90.537,400.482,165.373,54.989,159.762
C04305=1017.249,-90.287,400.473,165.377,54.982,159.762
C04306=1017.254,-90.037,400.464,165.379,54.977,159.761
C04307=1017.259,-89.788,400.455,165.382,54.971,159.761
C04308=1017.264,-89.537,400.446,165.385,54.965,159.761
C04309=1017.270,-89.288,400.436,165.388,54.960,159.760
C04310=1017.275,-89.038,400.428,165.392,54.954,159.760
C04311=1017.280,-88.788,400.419,165.395,54.948,159.760
C04312=1017.285,-88.539,400.410,165.397,54.943,159.759
C04313=1017.290,-88.288,400.400,165.400,54.937,159.759
C04314=1017.296,-88.039,400.392,165.403,54.931,159.759
C04315=1017.301,-87.790,400.383,165.407,54.925,159.759
C04316=1017.306,-87.540,400.373,165.410,54.920,159.758
C04317=1017.312,-87.290,400.364,165.412,54.913,159.758
C04318=1017.317,-87.040,400.355,165.415,54.908,159.757
C04319=1017.322,-86.790,400.346,165.419,54.902,159.757
C04320=1017.327,-86.541,400.337,165.421,54.896,159.757
C04321=1017.333,-86.290,400.328,165.424,54.891,159.756
C04322=1017.339,-86.010,400.318,165.428,54.884,159.756
C04323=1017.344,-85.729,400.307,165.431,54.877,159.755
C04324=1017.350,-85.448,400.297,165.435,54.871,159.755
C04325=1017.356,-85.167,400.287,165.438,54.865,159.755
C04326=1017.362,-84.918,400.277,165.441,54.859,159.754
C04327=1017.366,-84.668,400.268,165.443,54.853,159.754
C04328=1017.372,-84.418,400.259,165.446,54.847,159.753
C04329=1017.378,-84.168,400.250,165.450,54.841,159.753
C04330=1017.382,-83.919,400.240,165.453,54.835,159.753
C04331=1017.388,-83.669,400.232,165.456,54.830,159.753
C04332=1017.393,-83.419,400.221,165.459,54.824,159.752
C04333=1017.398,-83.169,400.213,165.462,54.817,159.752
C04334=1017.403,-82.920,400.203,165.465,54.812,159.751
C04335=1017.409,-82.669,400.194,165.468,54.806,159.751
C04336=1017.415,-82.420,400.185,165.471,54.800,159.751
C04337=1017.420,-82.171,400.175,165.474,54.794,159.750
C04338=1017.425,-81.920,400.166,165.477,54.788,159.750
C04339=1017.430,-81.671,400.157,165.479,54.783,159.749
C04340=1017.435,-81.421,400.148,165.483,54.777,159.749
C04341=1017.441,-81.171,400.138,165.486,54.770,159.749
C04342=1017.446,-80.921,400.129,165.488,54.765,159.748
C04343=1017.452,-80.671,400.119,165.492,54.759,159.748
C04344=1017.457,-80.422,400.110,165.495,54.753,159.748
C04345=1017.462,-80.172,400.101,165.498,54.748,159.747
C04346=1017.468,-79.922,400.091,165.500,54.741,159.747
C04347=1017.473,-79.673,400.082,165.503,54.736,159.746
C04348=1017.478,-79.423,400.072,165.507,54.730,159.746
C04349=1017.483,-79.173,400.062,165.510,54.724,159.746
C04350=1017.489,-78.923,400.053,165.513,54.719,159.745
C04351=1017.494,-78.674,400.043,165.515,54.713,159.745
C04352=1017.499,-78.424,400.033,165.518,54.708,159.745
C04353=1017.505,-78.174,400.024,165.522,54.702,159.744
C04354=1017.509,-77.924,400.015,165.525,54.696,159.744
C04355=1017.515,-77.674,400.004,165.528,54.690,159.744
C04356=1017.519,-77.425,399.995,165.531,54.685,159.743
C04357=1017.526,-77.175,399.985,165.533,54.678,159.743
C04358=1017.530,-76.926,399.975,165.537,54.673,159.743
C04359=1017.536,-76.676,399.965,165.540,54.667,159.742
C04360=1017.541,-76.426,399.957,165.543,54.661,159.742
C04361=1017.547,-76.176,399.946,165.545,54.656,159.741
C04362=1017.551,-75.926,399.937,165.548,54.650,159.741
C04363=1017.557,-75.676,399.927,165.552,54.644,159.741
C04364=1017.562,-75.427,399.917,165.554,54.638,159.740
C04365=1017.568,-75.177,399.907,165.557,54.632,159.740
C04366=1017.573,-74.928,399.897,165.560,54.627,159.739
C04367=1017.578,-74.677,399.887,165.563,54.621,159.739
C04368=1017.584,-74.428,399.878,165.567,54.615,159.739
C04369=1017.589,-74.178,399.868,165.570,54.610,159.739
C04370=1017.594,-73.929,399.858,165.573,54.604,159.738
C04371=1017.599,-73.679,399.848,165.575,54.599,159.738
C04372=1017.604,-73.429,399.838,165.578,54.593,159.737
C04373=1017.610,-73.179,399.828,165.581,54.587,159.737
C04374=1017.614,-72.929,399.817,165.584,54.582,159.737
C04375=1017.619,-72.679,399.807,165.587,54.576,159.736
C04376=1017.625,-72.429,399.797,165.590,54.571,159.736
C04377=1017.629,-72.180,399.787,165.592,54.565,159.736
C04378=1017.635,-71.930,399.777,165.596,54.559,159.735
C04379=1017.640,-71.681,399.767,165.599,54.554,159.735
C04380=1017.645,-71.431,399.757,165.602,54.548,159.735
C04381=1017.650,-71.181,399.747,165.605,54.542,159.734
C04382=1017.656,-70.931,399.737,165.608,54.537,159.734
C04383=1017.661,-70.681,399.726,165.611,54.531,159.733
C04384=1017.666,-70.432,399.717,165.613,54.526,159.733
C04385=1017.672,-70.182,399.706,165.616,54.520,159.733
C04386=1017.678,-69.904,399.695,165.620,54.514,159.732
C04387=1017.683,-69.625,399.683,165.624,54.508,159.732
C04388=1017.689,-69.346,399.672,165.626,54.501,159.731
C04389=1017.695,-69.067,399.660,165.629,54.495,159.731
C04390=1017.700,-68.817,399.650,165.632,54.489,159.731
C04391=1017.706,-68.567,399.640,165.635,54.483,159.730
C04392=1017.711,-68.318,399.630,165.639,54.478,159.730
C04393=1017.716,-68.068,399.620,165.642,54.472,159.730
C04394=1017.722,-67.818,399.609,165.645,54.466,159.729
C04395=1017.727,-67.569,399.599,165.647,54.461,159.729
C04396=1017.732,-67.319,399.589,165.650,54.455,159.729
C04397=1017.738,-67.069,399.578,165.653,54.450,159.728
C04398=1017.743,-66.820,399.569,165.656,54.444,159.728
C04399=1017.748,-66.570,399.558,165.660,54.438,159.728
C04400=1017.753,-66.320,399.548,165.662,54.432,159.727
C04401=1017.759,-66.070,399.537,165.665,54.426,159.727
C04402=1017.764,-65.821,399.528,165.668,54.421,159.726
C04403=1017.769,-65.571,399.517,165.671,54.415,159.726
C04404=1017.775,-65.321,399.507,165.674,54.410,159.725
C04405=1017.779,-65.071,399.496,165.678,54.404,159.725
C04406=1017.785,-64.821,399.486,165.680,54.398,159.725
C04407=1017.790,-64.572,399.475,165.683,54.392,159.724
C04408=1017.796,-64.322,399.465,165.686,54.386,159.724
C04409=1017.801,-64.072,399.455,165.689,54.381,159.724
C04410=1017.806,-63.823,399.444,165.691,54.375,159.723
C04411=1017.812,-63.573,399.434,165.695,54.369,159.723
C04412=1017.818,-63.323,399.423,165.698,54.363,159.722
C04413=1017.822,-63.074,399.413,165.701,54.358,159.722
C04414=1017.828,-62.824,399.403,165.703,54.352,159.722
C04415=1017.834,-62.574,399.392,165.706,54.347,159.721
C04416=1017.839,-62.324,399.382,165.710,54.341,159.721
C04417=1017.844,-62.075,399.372,165.713,54.334,159.720
C04418=1017.850,-61.825,399.362,165.715,54.329,159.720
C04419=1017.855,-61.575,399.351,165.718,54.323,159.720
C04420=1017.861,-61.326,399.341,165.721,54.318,159.719
C04421=1017.866,-61.075,399.330,165.724,54.311,159.719
C04422=1017.871,-60.826,399.319,165.727,54.306,159.718
C04423=1017.876,-60.576,399.309,165.730,54.300,159.718
C04424=1017.882,-60.327,399.298,165.733,54.294,159.718
C04425=1017.887,-60.077,399.288,165.736,54.288,159.717
C04426=1017.893,-59.827,399.277,165.738,54.283,159.717
C04427=1017.898,-59.577,399.267,165.742,54.277,159.716
C04428=1017.904,-59.328,399.256,165.745,54.271,159.716
C04429=1017.909,-59.078,399.246,165.748,54.265,159.715
C04430=1017.915,-58.829,399.236,165.751,54.259,159.715
C04431=1017.920,-58.579,399.225,165.754,54.253,159.715
C04432=1017.926,-58.329,399.214,165.757,54.247,159.714
C04433=1017.931,-58.079,399.204,165.760,54.242,159.714
C04434=1017.937,-57.829,399.193,165.763,54.236,159.713
C04435=1017.942,-57.579,399.183,165.765,54.230,159.713
C04436=1017.947,-57.330,399.172,165.769,54.224,159.713
C04437=1017.953,-57.081,399.161,165.772,54.218,159.712
C04438=1017.958,-56.831,399.151,165.774,54.212,159.712
C04439=1017.964,-56.581,399.140,165.777,54.207,159.711
C04440=1017.969,-56.331,399.130,165.781,54.201,159.711
C04441=1017.975,-56.082,399.119,165.783,54.194,159.710
C04442=1017.981,-55.832,399.108,165.786,54.189,159.710
C04443=1017.986,-55.582,399.098,165.789,54.183,159.710
C04444=1017.992,-55.332,399.087,165.791,54.177,159.709
C04445=1017.997,-55.082,399.077,165.795,54.171,159.709
C04446=1018.003,-54.833,399.066,165.798,54.166,159.708
C04447=1018.008,-54.583,399.055,165.801,54.160,159.708
C04448=1018.013,-54.333,399.045,165.804,54.154,159.707
C04449=1018.019,-54.083,399.034,165.807,54.147,159.707
C04450=1018.025,-53.806,399.022,165.810,54.141,159.706
C04451=1018.031,-53.528,399.011,165.813,54.134,159.706
C04452=1018.038,-53.251,398.998,165.816,54.128,159.705
C04453=1018.045,-52.973,398.986,165.820,54.121,159.705
C04454=1018.049,-52.723,398.976,165.823,54.116,159.705
C04455=1018.055,-52.473,398.965,165.826,54.109,159.704
C04456=1018.061,-52.224,398.954,165.829,54.104,159.704
C04457=1018.067,-51.974,398.943,165.832,54.098,159.703
C04458=1018.072,-51.724,398.933,165.834,54.092,159.703
C04459=1018.078,-51.475,398.922,165.838,54.086,159.702
C04460=1018.083,-51.225,398.911,165.841,54.080,159.702
C04461=1018.089,-50.976,398.900,165.844,54.074,159.701
C04462=1018.094,-50.725,398.889,165.846,54.069,159.701
C04463=1018.100,-50.476,398.878,165.849,54.062,159.700
C04464=1018.105,-50.226,398.867,165.852,54.057,159.700
C04465=1018.110,-49.976,398.856,165.855,54.051,159.700
C04466=1018.115,-49.727,398.845,165.859,54.046,159.699
C04467=1018.121,-49.477,398.834,165.861,54.040,159.699
C04468=1018.126,-49.227,398.822,165.864,54.034,159.699
C04469=1018.132,-48.978,398.811,165.867,54.028,159.698
C04470=1018.137,-48.728,398.800,165.870,54.023,159.698
C04471=1018.143,-48.479,398.789,165.873,54.017,159.697
C04472=1018.148,-48.229,398.778,165.875,54.012,159.697
C04473=1018.153,-47.979,398.767,165.878,54.006,159.696
C04474=1018.158,-47.729,398.755,165.881,54.000,159.696
C04475=1018.164,-47.480,398.744,165.884,53.994,159.695
C04476=1018.170,-47.229,398.733,165.888,53.989,159.695
C04477=1018.175,-46.980,398.722,165.890,53.983,159.695
C04478=1018.180,-46.730,398.710,165.893,53.977,159.694
C04479=1018.186,-46.481,398.699,165.896,53.971,159.694
C04480=1018.191,-46.231,398.687,165.899,53.966,159.693
C04481=1018.197,-45.982,398.676,165.901,53.960,159.693
C04482=1018.202,-45.732,398.665,165.904,53.954,159.692
C04483=1018.208,-45.483,398.654,165.907,53.949,159.692
C04484=1018.213,-45.233,398.642,165.911,53.943,159.692
C04485=1018.219,-44.983,398.631,165.913,53.937,159.691
C04486=1018.224,-44.733,398.620,165.916,53.931,159.691
C04487=1018.230,-44.483,398.609,165.919,53.926,159.690
C04488=1018.235,-44.234,398.597,165.921,53.919,159.690
C04489=1018.241,-43.985,398.586,165.924,53.914,159.689
C04490=1018.246,-43.735,398.574,165.927,53.908,159.689
C04491=1018.252,-43.484,398.562,165.930,53.902,159.688
C04492=1018.257,-43.235,398.552,165.934,53.896,159.688
C04493=1018.262,-42.985,398.540,165.937,53.891,159.688
C04494=1018.268,-42.736,398.529,165.939,53.885,159.687
C04495=1018.273,-42.486,398.517,165.942,53.879,159.687
C04496=1018.280,-42.236,398.506,165.945,53.874,159.686
C04497=1018.285,-41.986,398.494,165.947,53.867,159.686
C04498=1018.291,-41.737,398.483,165.950,53.862,159.685
C04499=1018.296,-41.487,398.472,165.954,53.856,159.685
C04500=1018.302,-41.238,398.460,165.957,53.850,159.685
C04501=1018.307,-40.988,398.449,165.959,53.844,159.684
C04502=1018.313,-40.738,398.438,165.962,53.839,159.684
C04503=1018.318,-40.489,398.426,165.965,53.833,159.683
C04504=1018.324,-40.239,398.415,165.968,53.827,159.683
C04505=1018.330,-39.989,398.403,165.971,53.821,159.682
C04506=1018.337,-39.629,398.386,165.975,53.813,159.682
C04507=1018.345,-39.268,398.369,165.979,53.804,159.681
C04508=1018.353,-38.907,398.353,165.984,53.796,159.680
C04509=1018.361,-38.546,398.336,165.988,53.788,159.680
C04510=1018.370,-38.130,398.317,165.992,53.779,159.679
C04511=1018.379,-37.714,398.297,165.997,53.769,159.678
C04512=1018.388,-37.298,398.277,166.001,53.759,159.677
C04513=1018.397,-36.882,398.258,166.007,53.750,159.677
C04514=1018.403,-36.632,398.245,166.009,53.744,159.676
C04515=1018.408,-36.383,398.234,166.012,53.738,159.676
C04516=1018.414,-36.133,398.222,166.015,53.733,159.675
C04517=1018.420,-35.883,398.210,166.018,53.727,159.675
C04518=1018.425,-35.634,398.198,166.021,53.721,159.674
C04519=1018.430,-35.384,398.187,166.024,53.716,159.674
C04520=1018.436,-35.134,398.174,166.026,53.710,159.674
C04521=1018.441,-34.885,398.163,166.029,53.704,159.673
C04522=1018.447,-34.636,398.151,166.032,53.699,159.673
C04523=1018.453,-34.385,398.139,166.036,53.693,159.672
C04524=1018.458,-34.136,398.127,166.038,53.687,159.672
C04525=1018.463,-33.886,398.116,166.041,53.681,159.671
C04526=1018.469,-33.636,398.103,166.044,53.676,159.671
C04527=1018.475,-33.387,398.092,166.047,53.669,159.670
C04528=1018.480,-33.138,398.080,166.049,53.664,159.670
C04529=1018.486,-32.887,398.068,166.052,53.659,159.670
C04530=1018.491,-32.638,398.056,166.055,53.652,159.669
C04531=1018.497,-32.388,398.044,166.058,53.647,159.669
C04532=1018.503,-32.139,398.033,166.060,53.641,159.668
C04533=1018.508,-31.889,398.020,166.063,53.635,159.668
C04534=1018.514,-31.639,398.009,166.066,53.630,159.667
C04535=1018.519,-31.390,397.996,166.070,53.623,159.667
C04536=1018.525,-31.140,397.984,166.073,53.618,159.666
C04537=1018.530,-30.890,397.972,166.075,53.612,159.666
C04538=1018.536,-30.641,397.961,166.078,53.606,159.665
C04539=1018.542,-30.391,397.948,166.081,53.601,159.665
C04540=1018.547,-30.142,397.937,166.083,53.594,159.664
C04541=1018.553,-29.892,397.924,166.086,53.589,159.664
C04542=1018.558,-29.642,397.913,166.089,53.583,159.663
C04543=1018.564,-29.392,397.901,166.092,53.577,159.663
C04544=1018.570,-29.143,397.889,166.095,53.571,159.662
C04545=1018.575,-28.893,397.876,166.098,53.565,159.662
C04546=1018.580,-28.643,397.865,166.101,53.559,159.661
C04547=1018.586,-28.394,397.852,166.104,53.554,159.661
C04548=1018.592,-28.144,397.840,166.106,53.548,159.661
C04549=1018.597,-27.895,397.829,166.109,53.542,159.660
C04550=1018.603,-27.645,397.816,166.112,53.537,159.660
C04551=1018.609,-27.396,397.804,166.114,53.530,159.659
C04552=1018.615,-27.146,397.792,166.117,53.525,159.659
C04553=1018.619,-26.895,397.779,166.120,53.520,159.658
C04554=1018.625,-26.646,397.767,166.123,53.513,159.657
C04555=1018.631,-26.396,397.754,166.126,53.508,159.657
C04556=1018.636,-26.147,397.742,166.129,53.502,159.657
C04557=1018.642,-25.897,397.730,166.131,53.497,159.656
C04558=1018.647,-25.648,397.718,166.134,53.491,159.656
C04559=1018.653,-25.398,397.705,166.137,53.485,159.655
C04560=1018.658,-25.149,397.693,166.140,53.480,159.655
C04561=1018.664,-24.899,397.680,166.142,53.474,159.654
C04562=1018.669,-24.649,397.667,166.145,53.468,159.654
C04563=1018.674,-24.399,397.656,166.148,53.463,159.653
C04564=1018.680,-24.150,397.643,166.151,53.457,159.653
C04565=1018.686,-23.900,397.631,166.154,53.451,159.652
C04566=1018.691,-23.651,397.619,166.156,53.445,159.652
C04567=1018.697,-23.401,397.606,166.159,53.440,159.651
C04568=1018.702,-23.151,397.594,166.163,53.434,159.651
C04569=1018.708,-22.902,397.581,166.166,53.428,159.651
C04570=1018.714,-22.652,397.569,166.168,53.422,159.650
C04571=1018.719,-22.403,397.557,166.171,53.417,159.650
C04572=1018.724,-22.152,397.544,166.174,53.411,159.649
C04573=1018.730,-21.903,397.531,166.177,53.405,159.649
C04574=1018.736,-21.625,397.518,166.179,53.399,159.648
C04575=1018.743,-21.347,397.503,166.183,53.393,159.648
C04576=1018.749,-21.068,397.490,166.186,53.386,159.647
C04577=1018.755,-20.790,397.476,166.189,53.380,159.646
C04578=1018.761,-20.540,397.463,166.191,53.374,159.646
C04579=1018.766,-20.291,397.451,166.194,53.368,159.645
C04580=1018.772,-20.041,397.438,166.197,53.362,159.645
C04581=1018.777,-19.792,397.426,166.200,53.357,159.644
C04582=1018.783,-19.541,397.413,166.202,53.351,159.644
C04583=1018.789,-19.292,397.400,166.205,53.345,159.643
C04584=1018.794,-19.043,397.388,166.209,53.339,159.643
C04585=1018.800,-18.793,397.375,166.212,53.333,159.643
C04586=1018.806,-18.543,397.362,166.214,53.327,159.642
C04587=1018.811,-18.294,397.350,166.217,53.322,159.641
C04588=1018.817,-18.044,397.338,166.220,53.315,159.641
C04589=1018.823,-17.794,397.325,166.223,53.310,159.640
C04590=1018.828,-17.545,397.312,166.225,53.304,159.640
C04591=1018.834,-17.295,397.300,166.228,53.298,159.639
C04592=1018.839,-17.045,397.287,166.231,53.292,159.639
C04593=1018.845,-16.796,397.274,166.234,53.287,159.638
C04594=1018.851,-16.547,397.262,166.236,53.281,159.638
C04595=1018.857,-16.297,397.249,166.239,53.275,159.637
C04596=1018.862,-16.048,397.237,166.242,53.269,159.637
C04597=1018.867,-15.797,397.224,166.245,53.264,159.636
C04598=1018.874,-15.548,397.211,166.247,53.258,159.636
C04599=1018.880,-15.298,397.198,166.250,53.252,159.635
C04600=1018.884,-15.049,397.185,166.253,53.247,159.635
C04601=1018.890,-14.799,397.172,166.255,53.241,159.634
C04602=1018.895,-14.549,397.159,166.258,53.235,159.634
C04603=1018.901,-14.300,397.147,166.261,53.230,159.633
C04604=1018.907,-14.050,397.134,166.264,53.224,159.633
C04605=1018.912,-13.801,397.120,166.267,53.218,159.632
C04606=1018.918,-13.551,397.108,166.269,53.212,159.632
C04607=1018.923,-13.302,397.094,166.272,53.207,159.631
C04608=1018.929,-13.052,397.082,166.275,53.201,159.631
C04609=1018.935,-12.802,397.069,166.278,53.195,159.630
C04610=1018.940,-12.553,397.055,166.281,53.190,159.630
C04611=1018.946,-12.303,397.043,166.283,53.184,159.629
C04612=1018.951,-12.053,397.030,166.286,53.178,159.629
C04613=1018.957,-11.804,397.017,166.289,53.172,159.628
C04614=1018.963,-11.554,397.004,166.292,53.167,159.628
C04615=1018.968,-11.305,396.991,166.295,53.161,159.627
C04616=1018.974,-11.055,396.978,166.297,53.155,159.627
C04617=1018.979,-10.805,396.965,166.300,53.150,159.626
C04618=1018.985,-10.556,396.952,166.303,53.144,159.626
C04619=1018.991,-10.306,396.939,166.306,53.138,159.625
C04620=1018.996,-10.057,396.926,166.308,53.132,159.625
C04621=1019.002,-9.807,396.913,166.311,53.127,159.624
C04622=1019.007,-9.558,396.899,166.314,53.121,159.624
C04623=1019.013,-9.308,396.887,166.317,53.115,159.623
C04624=1019.019,-9.058,396.873,166.319,53.109,159.623
C04625=1019.024,-8.809,396.861,166.322,53.104,159.622
C04626=1019.030,-8.560,396.847,166.325,53.098,159.622
C04627=1019.035,-8.309,396.834,166.328,53.092,159.621
C04628=1019.041,-8.060,396.821,166.330,53.086,159.621
C04629=1019.047,-7.810,396.808,166.333,53.081,159.620
C04630=1019.053,-7.561,396.794,166.336,53.074,159.620
C04631=1019.058,-7.312,396.782,166.339,53.069,159.619
C04632=1019.064,-7.062,396.768,166.341,53.063,159.619
C04633=1019.070,-6.812,396.756,166.344,53.057,159.618
C04634=1019.075,-6.563,396.742,166.347,53.051,159.618
C04635=1019.081,-6.313,396.729,166.349,53.045,159.617
C04636=1019.086,-6.063,396.716,166.352,53.040,159.616
C04637=1019.092,-5.813,396.703,166.355,53.034,159.616
C04638=1019.098,-5.533,396.688,166.358,53.027,159.615
C04639=1019.105,-5.253,396.673,166.361,53.021,159.615
C04640=1019.111,-4.973,396.658,166.364,53.014,159.614
C04641=1019.118,-4.693,396.644,166.367,53.008,159.613
C04642=1019.124,-4.444,396.631,166.369,53.002,159.613
C04643=1019.129,-4.194,396.617,166.372,52.996,159.612
C04644=1019.134,-3.944,396.604,166.375,52.991,159.612
C04645=1019.140,-3.694,396.590,166.378,52.985,159.611
C04646=1019.146,-3.445,396.577,166.381,52.980,159.611
C04647=1019.152,-3.196,396.563,166.383,52.973,159.610
C04648=1019.157,-2.945,396.550,166.386,52.968,159.610
C04649=1019.162,-2.696,396.536,166.389,52.963,159.609
C04650=1019.168,-2.446,396.522,166.392,52.957,159.609
C04651=1019.173,-2.198,396.509,166.395,52.951,159.608
C04652=1019.179,-1.948,396.495,166.396,52.945,159.608
C04653=1019.184,-1.699,396.481,166.399,52.940,159.607
C04654=1019.189,-1.448,396.468,166.402,52.935,159.607
C04655=1019.195,-1.199,396.454,166.405,52.929,159.606
C04656=1019.201,-0.949,396.441,166.408,52.923,159.606
C04657=1019.207,-0.700,396.427,166.410,52.917,159.605
C04658=1019.212,-0.450,396.413,166.413,52.912,159.605
C04659=1019.218,-0.201,396.399,166.416,52.906,159.604
C04660=1019.223,0.049,396.386,166.419,52.900,159.604
C04661=1019.229,0.299,396.373,166.422,52.895,159.603
C04662=1019.234,0.548,396.359,166.423,52.889,159.603
C04663=1019.240,0.798,396.345,166.426,52.884,159.602
C04664=1019.245,1.047,396.331,166.429,52.878,159.601
C04665=1019.251,1.297,396.318,166.432,52.872,159.601
C04666=1019.257,1.546,396.304,166.434,52.866,159.600
C04667=1019.263,1.796,396.290,166.437,52.861,159.600
C04668=1019.268,2.045,396.277,166.440,52.855,159.599
C04669=1019.274,2.295,396.263,166.443,52.849,159.599
C04670=1019.279,2.545,396.249,166.446,52.843,159.598
C04671=1019.285,2.794,396.236,166.449,52.838,159.598
C04672=1019.290,3.044,396.222,166.451,52.832,159.597
C04673=1019.296,3.294,396.209,166.454,52.826,159.597
C04674=1019.301,3.543,396.195,166.457,52.820,159.596
C04675=1019.307,3.793,396.181,166.459,52.815,159.596
C04676=1019.313,4.042,396.168,166.461,52.809,159.595
C04677=1019.318,4.292,396.154,166.464,52.803,159.594
C04678=1019.324,4.541,396.140,166.467,52.798,159.594
C04679=1019.329,4.791,396.126,166.469,52.792,159.593
C04680=1019.335,5.040,396.112,166.472,52.786,159.593
C04681=1019.341,5.290,396.099,166.475,52.780,159.592
C04682=1019.347,5.539,396.085,166.478,52.775,159.592
C04683=1019.352,5.789,396.071,166.480,52.769,159.591
C04684=1019.358,6.039,396.057,166.483,52.763,159.591
C04685=1019.364,6.289,396.043,166.486,52.757,159.590
C04686=1019.370,6.538,396.030,166.489,52.751,159.590
C04687=1019.375,6.787,396.016,166.492,52.746,159.589
C04688=1019.381,7.036,396.001,166.494,52.740,159.589
C04689=1019.387,7.286,395.987,166.497,52.734,159.588
C04690=1019.392,7.536,395.974,166.500,52.728,159.588
C04691=1019.398,7.785,395.960,166.502,52.722,159.587
C04692=1019.404,8.034,395.946,166.505,52.716,159.586
C04693=1019.409,8.284,395.933,166.507,52.711,159.586
C04694=1019.415,8.534,395.918,166.509,52.705,159.585
C04695=1019.421,8.784,395.905,166.512,52.699,159.584
C04696=1019.426,9.033,395.891,166.515,52.694,159.584
C04697=1019.432,9.283,395.877,166.518,52.688,159.583
C04698=1019.438,9.532,395.864,166.520,52.682,159.583
C04699=1019.444,9.781,395.849,166.523,52.676,159.582
C04700=1019.449,10.031,395.835,166.526,52.670,159.582
C04701=1019.455,10.281,395.821,166.528,52.664,159.581
C04702=1019.462,10.563,395.806,166.532,52.658,159.581
C04703=1019.468,10.845,395.790,166.534,52.651,159.580
C04704=1019.475,11.127,395.774,166.538,52.645,159.579
C04705=1019.481,11.409,395.758,166.541,52.638,159.579
C04706=1019.487,11.658,395.745,166.544,52.632,159.578
C04707=1019.493,11.909,395.730,166.547,52.626,159.577
C04708=1019.499,12.157,395.716,166.549,52.620,159.577
C04709=1019.504,12.407,395.702,166.552,52.615,159.576
C04710=1019.510,12.656,395.689,166.555,52.609,159.576
C04711=1019.516,12.906,395.675,166.557,52.603,159.575
C04712=1019.522,13.156,395.661,166.560,52.596,159.575
C04713=1019.528,13.405,395.646,166.563,52.591,159.574
C04714=1019.533,13.655,395.632,166.565,52.585,159.573
C04715=1019.539,13.904,395.618,166.567,52.579,159.573
C04716=1019.544,14.153,395.604,166.570,52.574,159.572
C04717=1019.550,14.404,395.589,166.573,52.568,159.572
C04718=1019.555,14.653,395.575,166.576,52.563,159.571
C04719=1019.561,14.902,395.560,166.578,52.557,159.571
C04720=1019.566,15.152,395.547,166.581,52.551,159.570
C04721=1019.572,15.402,395.533,166.584,52.545,159.570
C04722=1019.578,15.651,395.518,166.587,52.539,159.569
C04723=1019.584,15.901,395.504,166.589,52.533,159.568
C04724=1019.589,16.150,395.489,166.591,52.528,159.568
C04725=1019.595,16.399,395.475,166.594,52.522,159.567
C04726=1019.601,16.649,395.460,166.597,52.517,159.567
C04727=1019.606,16.899,395.446,166.599,52.511,159.566
C04728=1019.612,17.148,395.432,166.602,52.505,159.565
C04729=1019.617,17.397,395.418,166.605,52.499,159.565
C04730=1019.623,17.648,395.403,166.608,52.493,159.564
C04731=1019.629,17.897,395.389,166.610,52.487,159.564
C04732=1019.635,18.146,395.375,166.613,52.481,159.563
C04733=1019.641,18.396,395.360,166.616,52.476,159.563
C04734=1019.647,18.645,395.346,166.618,52.470,159.562
C04735=1019.652,18.895,395.331,166.621,52.464,159.561
C04736=1019.657,19.144,395.317,166.624,52.458,159.561
C04737=1019.663,19.394,395.302,166.626,52.453,159.560
C04738=1019.669,19.643,395.288,166.628,52.447,159.560
C04739=1019.675,19.892,395.274,166.631,52.441,159.559
C04740=1019.680,20.143,395.259,166.634,52.435,159.559
C04741=1019.686,20.392,395.244,166.637,52.429,159.558
C04742=1019.692,20.641,395.230,166.640,52.424,159.557
C04743=1019.697,20.892,395.215,166.642,52.418,159.557
C04744=1019.703,21.140,395.200,166.645,52.412,159.556
C04745=1019.708,21.390,395.186,166.648,52.407,159.556
C04746=1019.715,21.640,395.171,166.649,52.401,159.555
C04747=1019.720,21.889,395.156,166.652,52.395,159.554
C04748=1019.725,22.139,395.142,166.655,52.389,159.554
C04749=1019.731,22.388,395.127,166.658,52.384,159.553
C04750=1019.737,22.638,395.114,166.660,52.378,159.553
C04751=1019.742,22.887,395.098,166.663,52.372,159.552
C04752=1019.748,23.137,395.084,166.666,52.366,159.552
C04753=1019.754,23.386,395.070,166.669,52.360,159.551
C04754=1019.759,23.636,395.054,166.671,52.354,159.550
C04755=1019.765,23.885,395.040,166.674,52.348,159.550
C04756=1019.771,24.135,395.026,166.677,52.343,159.549
C04757=1019.777,24.384,395.011,166.678,52.337,159.549
C04758=1019.782,24.634,394.996,166.681,52.331,159.548
C04759=1019.788,24.883,394.982,166.684,52.325,159.547
C04760=1019.794,25.133,394.967,166.687,52.320,159.547
C04761=1019.799,25.382,394.952,166.689,52.314,159.546
C04762=1019.805,25.631,394.937,166.692,52.308,159.546
C04763=1019.811,25.881,394.923,166.695,52.302,159.545
C04764=1019.816,26.131,394.908,166.697,52.296,159.544
C04765=1019.822,26.380,394.893,166.700,52.290,159.544
C04766=1019.828,26.663,394.876,166.703,52.284,159.543
C04767=1019.835,26.947,394.860,166.706,52.277,159.542
C04768=1019.842,27.231,394.843,166.709,52.270,159.542
C04769=1019.848,27.514,394.826,166.712,52.263,159.541
C04770=1019.854,27.763,394.811,166.715,52.258,159.540
C04771=1019.859,28.013,394.796,166.717,52.252,159.540
C04772=1019.865,28.262,394.781,166.720,52.246,159.539
C04773=1019.871,28.512,394.766,166.723,52.240,159.539
C04774=1019.876,28.762,394.752,166.726,52.235,159.538
C04775=1019.882,29.012,394.736,166.727,52.229,159.537
C04776=1019.887,29.261,394.721,166.730,52.223,159.537
C04777=1019.893,29.511,394.706,166.733,52.218,159.536
C04778=1019.898,29.760,394.691,166.736,52.212,159.536
C04779=1019.904,30.009,394.676,166.738,52.206,159.535
C04780=1019.910,30.259,394.661,166.741,52.200,159.534
C04781=1019.916,30.508,394.646,166.744,52.195,159.534
C04782=1019.921,30.758,394.631,166.747,52.189,159.533
C04783=1019.927,31.007,394.616,166.748,52.183,159.533
C04784=1019.933,31.257,394.600,166.751,52.177,159.532
C04785=1019.938,31.506,394.586,166.754,52.172,159.532
C04786=1019.944,31.756,394.570,166.756,52.166,159.531
C04787=1019.950,32.005,394.556,166.759,52.160,159.530
C04788=1019.955,32.255,394.540,166.762,52.154,159.530
C04789=1019.961,32.504,394.526,166.764,52.148,159.529
C04790=1019.967,32.754,394.510,166.767,52.142,159.529
C04791=1019.973,33.003,394.496,166.770,52.136,159.528
C04792=1019.978,33.253,394.480,166.773,52.130,159.527
C04793=1019.983,33.502,394.465,166.774,52.125,159.527
C04794=1019.990,33.751,394.450,166.777,52.119,159.526
C04795=1019.995,34.001,394.435,166.780,52.113,159.525
C04796=1020.001,34.250,394.420,166.782,52.107,159.525
C04797=1020.006,34.500,394.405,166.785,52.101,159.524
C04798=1020.013,34.749,394.390,166.788,52.095,159.524
C04799=1020.018,34.999,394.374,166.791,52.089,159.523
C04800=1020.024,35.248,394.360,166.793,52.083,159.522
C04801=1020.029,35.497,394.344,166.796,52.077,159.522
C04802=1020.035,35.747,394.329,166.799,52.071,159.521
C04803=1020.041,35.997,394.314,166.801,52.065,159.520
C04804=1020.046,36.246,394.299,166.804,52.059,159.520
C04805=1020.052,36.496,394.284,166.807,52.054,159.519
C04806=1020.058,36.745,394.269,166.809,52.049,159.519
C04807=1020.063,36.995,394.252,166.811,52.043,159.518
C04808=1020.069,37.244,394.238,166.814,52.037,159.517
C04809=1020.075,37.494,394.222,166.817,52.031,159.517
C04810=1020.081,37.744,394.207,166.820,52.025,159.516
C04811=1020.086,37.993,394.191,166.822,52.019,159.516
C04812=1020.092,38.242,394.175,166.825,52.013,159.515
C04813=1020.097,38.491,394.161,166.827,52.008,159.514
C04814=1020.103,38.741,394.145,166.829,52.002,159.513
C04815=1020.109,38.991,394.130,166.832,51.996,159.513
C04816=1020.114,39.240,394.114,166.835,51.990,159.512
C04817=1020.120,39.489,394.099,166.838,51.984,159.512
C04818=1020.125,39.739,394.084,166.840,51.979,159.511
C04819=1020.131,39.989,394.068,166.843,51.973,159.510
C04820=1020.137,40.238,394.052,166.846,51.967,159.510
C04821=1020.142,40.487,394.037,166.848,51.962,159.509
C04822=1020.148,40.737,394.022,166.850,51.956,159.509
C04823=1020.154,40.985,394.006,166.853,51.950,159.508
C04824=1020.159,41.235,393.990,166.856,51.944,159.507
C04825=1020.165,41.485,393.975,166.858,51.938,159.507
C04826=1020.170,41.735,393.959,166.861,51.932,159.506
C04827=1020.177,41.984,393.944,166.864,51.926,159.506
C04828=1020.182,42.234,393.928,166.867,51.921,159.505
C04829=1020.187,42.483,393.913,166.870,51.915,159.504
C04830=1020.193,42.766,393.895,166.872,51.908,159.504
C04831=1020.200,43.050,393.877,166.874,51.902,159.503
C04832=1020.206,43.333,393.859,166.878,51.895,159.502
C04833=1020.213,43.617,393.841,166.880,51.889,159.502
C04834=1020.219,43.866,393.825,166.883,51.883,159.501
C04835=1020.224,44.116,393.809,166.886,51.877,159.500
C04836=1020.229,44.365,393.793,166.889,51.872,159.500
C04837=1020.234,44.615,393.777,166.892,51.866,159.499
C04838=1020.240,44.864,393.761,166.893,51.860,159.498
C04839=1020.245,45.113,393.746,166.896,51.854,159.498
C04840=1020.251,45.362,393.730,166.899,51.849,159.497
C04841=1020.257,45.612,393.714,166.902,51.843,159.497
C04842=1020.262,45.861,393.698,166.904,51.837,159.496
C04843=1020.268,46.111,393.683,166.907,51.831,159.495
C04844=1020.274,46.360,393.667,166.909,51.825,159.495
C04845=1020.280,46.610,393.651,166.912,51.820,159.494
C04846=1020.285,46.859,393.635,166.914,51.814,159.494
C04847=1020.291,47.109,393.620,166.917,51.808,159.493
C04848=1020.296,47.359,393.603,166.920,51.802,159.492
C04849=1020.301,47.607,393.587,166.923,51.796,159.492
C04850=1020.307,47.857,393.571,166.925,51.791,159.491
C04851=1020.313,48.107,393.555,166.927,51.786,159.490
C04852=1020.318,48.356,393.540,166.930,51.780,159.490
C04853=1020.324,48.605,393.524,166.933,51.774,159.489
C04854=1020.330,48.855,393.507,166.935,51.768,159.489
C04855=1020.335,49.105,393.492,166.938,51.762,159.488
C04856=1020.341,49.353,393.476,166.941,51.756,159.487
C04857=1020.346,49.603,393.460,166.943,51.751,159.487
C04858=1020.352,49.853,393.444,166.946,51.745,159.486
C04859=1020.358,50.102,393.427,166.948,51.739,159.485
C04860=1020.363,50.351,393.412,166.951,51.733,159.485
C04861=1020.369,50.601,393.396,166.954,51.727,159.484
C04862=1020.374,50.850,393.380,166.956,51.721,159.484
C04863=1020.380,51.100,393.364,166.959,51.715,159.483
C04864=1020.385,51.349,393.348,166.962,51.709,159.482
C04865=1020.391,51.598,393.332,166.963,51.704,159.481
C04866=1020.397,51.848,393.316,166.966,51.698,159.481
C04867=1020.403,52.097,393.300,166.969,51.692,159.480
C04868=1020.409,52.347,393.284,166.972,51.687,159.480
C04869=1020.414,52.596,393.267,166.975,51.681,159.479
C04870=1020.419,52.846,393.252,166.977,51.675,159.478
C04871=1020.425,53.095,393.236,166.980,51.669,159.478
C04872=1020.431,53.344,393.219,166.983,51.663,159.477
C04873=1020.437,53.594,393.204,166.985,51.657,159.477
C04874=1020.442,53.843,393.188,166.987,51.651,159.476
C04875=1020.448,54.092,393.172,166.990,51.645,159.475
C04876=1020.454,54.342,393.155,166.992,51.639,159.475
C04877=1020.460,54.592,393.140,166.995,51.633,159.474
C04878=1020.465,54.841,393.123,166.998,51.627,159.473
C04879=1020.471,55.091,393.107,167.001,51.622,159.473
C04880=1020.476,55.339,393.091,167.003,51.616,159.472
C04881=1020.482,55.589,393.075,167.006,51.610,159.471
C04882=1020.488,55.839,393.059,167.009,51.604,159.471
C04883=1020.494,56.088,393.043,167.011,51.598,159.470
C04884=1020.500,56.337,393.026,167.014,51.592,159.469
C04885=1020.506,56.587,393.010,167.017,51.586,159.469
C04886=1020.511,56.836,392.995,167.019,51.580,159.468
C04887=1020.516,57.086,392.978,167.021,51.574,159.467
C04888=1020.522,57.335,392.962,167.024,51.569,159.467
C04889=1020.528,57.584,392.946,167.027,51.563,159.466
C04890=1020.534,57.834,392.929,167.029,51.556,159.465
C04891=1020.539,58.084,392.914,167.032,51.550,159.465
C04892=1020.545,58.333,392.898,167.034,51.544,159.464
C04893=1020.551,58.582,392.881,167.037,51.538,159.463
C04894=1020.558,58.865,392.862,167.041,51.531,159.463
C04895=1020.564,59.148,392.845,167.043,51.525,159.462
C04896=1020.571,59.433,392.826,167.046,51.518,159.461
C04897=1020.578,59.715,392.808,167.050,51.511,159.460
C04898=1020.583,59.965,392.791,167.052,51.505,159.460
C04899=1020.588,60.215,392.775,167.054,51.499,159.459
C04900=1020.594,60.464,392.759,167.057,51.493,159.458
C04901=1020.600,60.713,392.743,167.059,51.487,159.458
C04902=1020.606,60.963,392.727,167.062,51.481,159.457
C04903=1020.612,61.212,392.710,167.065,51.476,159.456
C04904=1020.618,61.461,392.694,167.068,51.470,159.456
C04905=1020.624,61.710,392.678,167.070,51.463,159.455
C04906=1020.629,61.960,392.661,167.073,51.457,159.454
C04907=1020.635,62.209,392.645,167.075,51.451,159.453
C04908=1020.641,62.458,392.629,167.078,51.445,159.453
C04909=1020.647,62.708,392.613,167.081,51.439,159.452
C04910=1020.653,62.957,392.596,167.084,51.433,159.452
C04911=1020.658,63.207,392.579,167.086,51.428,159.451
C04912=1020.664,63.456,392.563,167.089,51.422,159.450
C04913=1020.670,63.705,392.547,167.092,51.416,159.450
C04914=1020.675,63.955,392.530,167.095,51.410,159.449
C04915=1020.681,64.205,392.514,167.097,51.404,159.448
C04916=1020.686,64.454,392.497,167.100,51.398,159.448
C04917=1020.692,64.704,392.481,167.102,51.392,159.447
C04918=1020.697,64.953,392.464,167.104,51.387,159.446
C04919=1020.703,65.203,392.448,167.107,51.381,159.446
C04920=1020.709,65.452,392.430,167.110,51.375,159.445
C04921=1020.715,65.701,392.414,167.112,51.368,159.444
C04922=1020.721,65.950,392.398,167.115,51.362,159.443
C04923=1020.726,66.200,392.381,167.118,51.356,159.443
C04924=1020.732,66.449,392.364,167.120,51.350,159.442
C04925=1020.737,66.699,392.348,167.123,51.345,159.442
C04926=1020.743,66.948,392.331,167.126,51.339,159.441
C04927=1020.748,67.197,392.314,167.128,51.333,159.440
C04928=1020.754,67.447,392.298,167.130,51.327,159.440
C04929=1020.760,67.696,392.281,167.133,51.321,159.439
C04930=1020.766,67.945,392.264,167.136,51.315,159.438
C04931=1020.771,68.195,392.247,167.139,51.310,159.438
C04932=1020.777,68.444,392.231,167.141,51.304,159.437
C04933=1020.782,68.694,392.214,167.144,51.298,159.436
C04934=1020.788,68.943,392.196,167.147,51.292,159.436
C04935=1020.794,69.192,392.180,167.150,51.286,159.435
C04936=1020.799,69.442,392.163,167.152,51.280,159.434
C04937=1020.805,69.690,392.146,167.154,51.275,159.434
C04938=1020.810,69.940,392.129,167.157,51.269,159.433
C04939=1020.816,70.190,392.112,167.160,51.263,159.432
C04940=1020.822,70.439,392.095,167.162,51.257,159.432
C04941=1020.827,70.688,392.079,167.165,51.251,159.431
C04942=1020.833,70.939,392.061,167.168,51.245,159.430
C04943=1020.839,71.187,392.044,167.171,51.239,159.430
C04944=1020.844,71.437,392.028,167.173,51.233,159.429
C04945=1020.850,71.687,392.011,167.176,51.227,159.428
C04946=1020.856,71.935,391.994,167.178,51.222,159.428
C04947=1020.861,72.185,391.977,167.181,51.216,159.427
C04948=1020.867,72.434,391.959,167.183,51.210,159.426
C04949=1020.873,72.683,391.943,167.186,51.204,159.426
C04950=1020.878,72.933,391.926,167.189,51.198,159.425
C04951=1020.883,73.182,391.909,167.192,51.193,159.424
C04952=1020.889,73.431,391.892,167.194,51.187,159.424
C04953=1020.895,73.680,391.875,167.197,51.181,159.423
C04954=1020.900,73.930,391.858,167.200,51.175,159.423
C04955=1020.907,74.180,391.841,167.202,51.168,159.422
C04956=1020.912,74.429,391.824,167.204,51.163,159.421
C04957=1020.917,74.679,391.807,167.207,51.157,159.420
C04958=1020.924,74.961,391.787,167.210,51.150,159.420
C04959=1020.931,75.245,391.768,167.214,51.143,159.419
C04960=1020.937,75.528,391.749,167.216,51.137,159.418
C04961=1020.944,75.811,391.730,167.220,51.130,159.417
C04962=1020.949,76.061,391.713,167.222,51.124,159.417
C04963=1020.954,76.310,391.695,167.225,51.118,159.416
C04964=1020.960,76.559,391.678,167.227,51.112,159.415
C04965=1020.966,76.809,391.660,167.230,51.107,159.415
C04966=1020.972,77.058,391.643,167.232,51.101,159.414
C04967=1020.977,77.308,391.627,167.235,51.095,159.413
C04968=1020.983,77.557,391.609,167.238,51.089,159.413
C04969=1020.988,77.806,391.592,167.241,51.083,159.412
C04970=1020.993,78.055,391.575,167.243,51.077,159.411
C04971=1020.999,78.304,391.557,167.246,51.071,159.411
C04972=1021.005,78.555,391.540,167.249,51.065,159.410
C04973=1021.010,78.804,391.522,167.251,51.060,159.409
C04974=1021.016,79.053,391.505,167.253,51.054,159.409
C04975=1021.021,79.302,391.488,167.256,51.048,159.408
C04976=1021.026,79.552,391.470,167.259,51.042,159.407
C04977=1021.032,79.801,391.453,167.262,51.037,159.407
C04978=1021.038,80.050,391.435,167.265,51.031,159.406
C04979=1021.043,80.300,391.418,167.267,51.025,159.405
C04980=1021.049,80.549,391.400,167.269,51.019,159.405
C04981=1021.054,80.798,391.383,167.272,51.013,159.404
C04982=1021.061,81.047,391.366,167.275,51.008,159.403
C04983=1021.066,81.296,391.349,167.277,51.002,159.403
C04984=1021.072,81.546,391.331,167.280,50.996,159.402
C04985=1021.077,81.795,391.313,167.283,50.990,159.401
C04986=1021.083,82.045,391.297,167.286,50.984,159.401
C04987=1021.088,82.294,391.279,167.289,50.978,159.400
C04988=1021.094,82.544,391.261,167.291,50.972,159.399
C04989=1021.100,82.793,391.243,167.294,50.967,159.399
C04990=1021.105,83.042,391.226,167.296,50.961,159.398
C04991=1021.111,83.291,391.209,167.299,50.955,159.397
C04992=1021.116,83.540,391.191,167.302,50.949,159.397
C04993=1021.122,83.790,391.174,167.304,50.944,159.396
C04994=1021.128,84.039,391.156,167.307,50.937,159.395
C04995=1021.133,84.288,391.138,167.310,50.931,159.395
C04996=1021.138,84.538,391.122,167.312,50.925,159.394
C04997=1021.145,84.788,391.104,167.315,50.920,159.393
C04998=1021.150,85.037,391.086,167.318,50.914,159.393
C04999=1021.156,85.286,391.069,167.321,50.908,159.392
C05000=1021.161,85.535,391.051,167.324,50.902,159.391
C05001=1021.167,85.785,391.033,167.326,50.896,159.391
C05002=1021.172,86.034,391.016,167.329,50.890,159.390
C05003=1021.178,86.283,390.999,167.332,50.884,159.389
C05004=1021.184,86.533,390.981,167.334,50.878,159.389
C05005=1021.190,86.782,390.963,167.336,50.872,159.388
C05006=1021.195,87.031,390.946,167.339,50.867,159.387
C05007=1021.201,87.280,390.928,167.342,50.861,159.387
C05008=1021.207,87.530,390.910,167.345,50.855,159.386
C05009=1021.212,87.779,390.892,167.347,50.848,159.385
C05010=1021.218,88.029,390.876,167.350,50.843,159.384
C05011=1021.224,88.278,390.858,167.353,50.837,159.384
C05012=1021.229,88.527,390.840,167.355,50.831,159.383
C05013=1021.235,88.776,390.823,167.358,50.825,159.382
C05014=1021.241,89.026,390.805,167.361,50.819,159.382
C05015=1021.246,89.275,390.787,167.363,50.813,159.381
C05016=1021.252,89.524,390.769,167.366,50.807,159.380
C05017=1021.257,89.774,390.751,167.369,50.801,159.380
C05018=1021.263,90.023,390.733,167.372,50.795,159.379
C05019=1021.268,90.272,390.716,167.375,50.789,159.378
C05020=1021.274,90.522,390.698,167.376,50.784,159.378
C05021=1021.279,90.771,390.679,167.379,50.778,159.377
C05022=1021.286,91.055,390.659,167.383,50.771,159.376
C05023=1021.293,91.338,390.639,167.387,50.765,159.376
C05024=1021.298,91.620,390.619,167.389,50.759,159.375
C05025=1021.305,91.903,390.598,167.392,50.752,159.374
C05026=1021.310,92.153,390.580,167.395,50.746,159.373
C05027=1021.316,92.402,390.562,167.397,50.740,159.373
C05028=1021.321,92.652,390.544,167.400,50.735,159.372
C05029=1021.327,92.901,390.526,167.403,50.729,159.371
C05030=1021.332,93.151,390.508,167.406,50.723,159.371
C05031=1021.338,93.399,390.490,167.408,50.717,159.370
C05032=1021.344,93.649,390.472,167.411,50.711,159.369
C05033=1021.349,93.898,390.454,167.414,50.705,159.369
C05034=1021.355,94.148,390.436,167.416,50.699,159.368
C05035=1021.360,94.397,390.418,167.419,50.693,159.367
C05036=1021.366,94.646,390.400,167.422,50.687,159.367
C05037=1021.372,94.895,390.382,167.425,50.682,159.366
C05038=1021.377,95.144,390.364,167.428,50.676,159.365
C05039=1021.383,95.394,390.346,167.431,50.670,159.365
C05040=1021.388,95.644,390.328,167.433,50.664,159.364
C05041=1021.394,95.892,390.310,167.436,50.658,159.363
C05042=1021.400,96.142,390.292,167.438,50.652,159.362
C05043=1021.405,96.391,390.274,167.440,50.646,159.362
C05044=1021.411,96.641,390.256,167.443,50.641,159.361
C05045=1021.417,96.889,390.237,167.446,50.635,159.360
C05046=1021.422,97.139,390.219,167.449,50.629,159.360
C05047=1021.428,97.388,390.201,167.452,50.623,159.359
C05048=1021.433,97.637,390.184,167.455,50.617,159.359
C05049=1021.439,97.887,390.164,167.457,50.611,159.358
C05050=1021.444,98.136,390.147,167.460,50.605,159.357
C05051=1021.451,98.386,390.129,167.463,50.599,159.356
C05052=1021.456,98.635,390.111,167.466,50.594,159.356
C05053=1021.462,98.884,390.092,167.468,50.588,159.355
C05054=1021.467,99.133,390.075,167.471,50.582,159.354
C05055=1021.473,99.383,390.057,167.474,50.575,159.354
C05056=1021.478,99.632,390.038,167.477,50.570,159.353
C05057=1021.484,99.882,390.019,167.479,50.564,159.352
C05058=1021.490,100.130,390.001,167.482,50.558,159.352
C05059=1021.494,100.379,389.983,167.485,50.552,159.351
C05060=1021.501,100.628,389.964,167.488,50.547,159.350
C05061=1021.506,100.878,389.946,167.491,50.541,159.350
C05062=1021.511,101.127,389.927,167.493,50.535,159.349
C05063=1021.517,101.376,389.909,167.495,50.529,159.348
C05064=1021.522,101.626,389.891,167.498,50.524,159.348
C05065=1021.528,101.875,389.872,167.501,50.518,159.347
C05066=1021.533,102.125,389.854,167.504,50.512,159.346
C05067=1021.539,102.374,389.835,167.507,50.506,159.346
C05068=1021.545,102.623,389.816,167.510,50.501,159.345
C05069=1021.550,102.872,389.798,167.513,50.495,159.344
C05070=1021.556,103.121,389.780,167.515,50.489,159.344
C05071=1021.561,103.370,389.761,167.518,50.483,159.343
C05072=1021.567,103.620,389.742,167.521,50.477,159.342
C05073=1021.572,103.869,389.725,167.524,50.472,159.342
C05074=1021.578,104.118,389.705,167.527,50.466,159.341
C05075=1021.583,104.367,389.688,167.529,50.459,159.340
C05076=1021.589,104.617,389.669,167.532,50.454,159.340
C05077=1021.594,104.866,389.650,167.535,50.448,159.339
C05078=1021.600,105.115,389.632,167.538,50.442,159.338
C05079=1021.605,105.364,389.613,167.540,50.437,159.338
C05080=1021.611,105.614,389.595,167.542,50.431,159.337
C05081=1021.617,105.863,389.576,167.545,50.425,159.336
C05082=1021.622,106.113,389.557,167.548,50.419,159.336
C05083=1021.628,106.362,389.539,167.551,50.413,159.335
C05084=1021.633,106.610,389.520,167.554,50.408,159.334
C05085=1021.639,106.860,389.501,167.556,50.401,159.333
C05086=1021.646,107.143,389.480,167.560,50.394,159.333
C05087=1021.652,107.426,389.459,167.563,50.388,159.332
C05088=1021.659,107.710,389.438,167.566,50.382,159.331
C05089=1021.665,107.994,389.417,167.570,50.375,159.331
C05090=1021.670,108.242,389.399,167.572,50.369,159.330
C05091=1021.676,108.492,389.380,167.575,50.363,159.329
C05092=1021.681,108.742,389.361,167.578,50.357,159.328
C05093=1021.687,108.990,389.343,167.581,50.351,159.328
C05094=1021.693,109.240,389.324,167.584,50.346,159.327
C05095=1021.698,109.489,389.305,167.587,50.340,159.327
C05096=1021.704,109.738,389.287,167.589,50.333,159.326
C05097=1021.710,109.988,389.268,167.592,50.328,159.325
C05098=1021.715,110.236,389.249,167.595,50.322,159.324
C05099=1021.721,110.486,389.229,167.598,50.316,159.324
C05100=1021.726,110.735,389.212,167.601,50.310,159.323
C05101=1021.732,110.984,389.193,167.603,50.305,159.322
C05102=1021.737,111.234,389.173,167.606,50.299,159.322
C05103=1021.743,111.482,389.154,167.609,50.293,159.321
C05104=1021.748,111.732,389.135,167.612,50.287,159.320
C05105=1021.754,111.982,389.117,167.615,50.282,159.320
C05106=1021.759,112.230,389.098,167.618,50.276,159.319
C05107=1021.765,112.480,389.079,167.621,50.270,159.319
C05108=1021.771,112.729,389.060,167.624,50.264,159.318
C05109=1021.776,112.978,389.041,167.626,50.259,159.317
C05110=1021.782,113.227,389.022,167.629,50.253,159.317
C05111=1021.787,113.477,389.003,167.632,50.247,159.316
C05112=1021.792,113.725,388.984,167.634,50.242,159.315
C05113=1021.797,113.975,388.964,167.637,50.236,159.314
C05114=1021.802,114.224,388.945,167.640,50.230,159.314
C05115=1021.808,114.473,388.926,167.643,50.224,159.313
C05116=1021.814,114.723,388.906,167.646,50.219,159.313
C05117=1021.819,114.972,388.888,167.649,50.213,159.312
C05118=1021.825,115.221,388.868,167.651,50.207,159.311
C05119=1021.830,115.470,388.849,167.654,50.201,159.311
C05120=1021.835,115.719,388.830,167.657,50.196,159.310
C05121=1021.841,115.969,388.811,167.660,50.190,159.309
C05122=1021.847,116.218,388.792,167.663,50.184,159.309
C05123=1021.852,116.467,388.773,167.666,50.178,159.308
C05124=1021.857,116.716,388.753,167.669,50.173,159.307
C05125=1021.862,116.966,388.734,167.672,50.167,159.307
C05126=1021.868,117.215,388.715,167.674,50.161,159.306
C05127=1021.874,117.463,388.695,167.677,50.155,159.305
C05128=1021.879,117.713,388.676,167.680,50.150,159.305
C05129=1021.885,117.962,388.656,167.683,50.144,159.304
C05130=1021.890,118.211,388.638,167.686,50.138,159.303
C05131=1021.896,118.460,388.618,167.689,50.133,159.303
C05132=1021.901,118.710,388.599,167.692,50.127,159.302
C05133=1021.907,118.959,388.580,167.695,50.121,159.301
C05134=1021.911,119.208,388.560,167.698,50.115,159.301
C05135=1021.917,119.458,388.541,167.701,50.110,159.300
C05136=1021.923,119.707,388.521,167.703,50.104,159.299
C05137=1021.928,119.955,388.502,167.706,50.098,159.299
C05138=1021.934,120.205,388.483,167.709,50.092,159.298
C05139=1021.940,120.454,388.464,167.712,50.087,159.298
C05140=1021.945,120.704,388.445,167.715,50.081,159.297
C05141=1021.951,120.953,388.425,167.718,50.075,159.296
C05142=1021.956,121.201,388.406,167.721,50.070,159.296
C05143=1021.962,121.451,388.387,167.724,50.064,159.295
C05144=1021.967,121.700,388.367,167.727,50.058,159.294
C05145=1021.973,121.950,388.347,167.730,50.052,159.294
C05146=1021.979,122.214,388.327,167.732,50.046,159.293
C05147=1021.985,122.478,388.306,167.735,50.040,159.292
C05148=1021.991,122.741,388.286,167.739,50.033,159.291
C05149=1021.996,123.006,388.265,167.741,50.028,159.291
C05150=1022.003,123.274,388.245,167.744,50.021,159.290
C05151=1022.008,123.542,388.224,167.748,50.015,159.289
C05152=1022.015,123.811,388.202,167.750,50.009,159.288
C05153=1022.020,124.079,388.182,167.754,50.003,159.288
C05154=1022.026,124.329,388.162,167.757,49.997,159.287
C05155=1022.032,124.578,388.142,167.760,49.991,159.287
C05156=1022.037,124.826,388.123,167.763,49.986,159.286
C05157=1022.043,125.076,388.104,167.766,49.979,159.285
C05158=1022.049,125.325,388.084,167.769,49.974,159.284
C05159=1022.054,125.574,388.065,167.771,49.968,159.284
C05160=1022.060,125.824,388.046,167.774,49.962,159.283
C05161=1022.065,126.073,388.025,167.777,49.957,159.282
C05162=1022.071,126.322,388.006,167.780,49.951,159.282
C05163=1022.076,126.571,387.987,167.784,49.945,159.281
C05164=1022.082,126.820,387.967,167.787,49.939,159.281
C05165=1022.088,127.069,387.948,167.790,49.933,159.280
C05166=1022.093,127.318,387.929,167.793,49.927,159.279
C05167=1022.099,127.567,387.909,167.795,49.921,159.278
C05168=1022.105,127.817,387.889,167.798,49.916,159.278
C05169=1022.110,128.066,387.870,167.801,49.910,159.277
C05170=1022.116,128.315,387.850,167.804,49.904,159.276
C05171=1022.122,128.565,387.830,167.807,49.898,159.276
C05172=1022.127,128.813,387.811,167.811,49.892,159.275
C05173=1022.133,129.062,387.792,167.814,49.886,159.274
C05174=1022.138,129.312,387.772,167.817,49.880,159.274
C05175=1022.144,129.560,387.752,167.820,49.875,159.273
C05176=1022.150,129.810,387.733,167.822,49.869,159.272
C05177=1022.155,130.059,387.713,167.825,49.863,159.272
C05178=1022.161,130.308,387.693,167.828,49.858,159.271
C05179=1022.166,130.558,387.673,167.831,49.852,159.270
C05180=1022.172,130.807,387.654,167.834,49.846,159.270
C05181=1022.177,131.056,387.633,167.837,49.840,159.269
C05182=1022.183,131.305,387.613,167.840,49.835,159.269
C05183=1022.189,131.554,387.594,167.843,49.829,159.268
C05184=1022.194,131.804,387.573,167.846,49.823,159.267
C05185=1022.199,132.052,387.554,167.850,49.817,159.267
C05186=1022.205,132.301,387.534,167.853,49.812,159.266
C05187=1022.211,132.550,387.514,167.856,49.806,159.265
C05188=1022.215,132.800,387.494,167.859,49.800,159.265
C05189=1022.221,133.049,387.474,167.862,49.795,159.264
C05190=1022.227,133.298,387.453,167.865,49.789,159.263
C05191=1022.232,133.547,387.434,167.867,49.783,159.263
C05192=1022.238,133.796,387.414,167.870,49.778,159.262
C05193=1022.244,134.045,387.394,167.873,49.772,159.261
C05194=1022.249,134.295,387.374,167.876,49.766,159.261
C05195=1022.255,134.544,387.354,167.879,49.761,159.260
C05196=1022.260,134.793,387.333,167.882,49.755,159.259
C05197=1022.266,135.042,387.313,167.886,49.749,159.259
C05198=1022.271,135.291,387.294,167.889,49.743,159.258
C05199=1022.277,135.540,387.274,167.892,49.738,159.258
C05200=1022.282,135.789,387.253,167.895,49.732,159.257
C05201=1022.288,136.039,387.234,167.898,49.726,159.256
C05202=1022.293,136.288,387.213,167.901,49.721,159.256
C05203=1022.299,136.537,387.193,167.904,49.715,159.255
C05204=1022.304,136.786,387.173,167.907,49.709,159.254
C05205=1022.310,137.035,387.153,167.910,49.703,159.254
C05206=1022.315,137.284,387.133,167.913,49.698,159.253
C05207=1022.321,137.533,387.113,167.917,49.692,159.252
C05208=1022.326,137.782,387.092,167.920,49.686,159.252
C05209=1022.332,138.032,387.072,167.922,49.680,159.251
C05210=1022.338,138.280,387.052,167.926,49.675,159.251
C05211=1022.343,138.529,387.031,167.929,49.670,159.250
C05212=1022.348,138.779,387.011,167.932,49.664,159.249
C05213=1022.354,139.028,386.992,167.935,49.658,159.249
C05214=1022.360,139.311,386.968,167.938,49.652,159.248
C05215=1022.366,139.595,386.944,167.942,49.645,159.247
C05216=1022.373,139.878,386.921,167.946,49.639,159.247
C05217=1022.379,140.161,386.898,167.948,49.633,159.246
C05218=1022.384,140.410,386.877,167.951,49.627,159.245
C05219=1022.390,140.659,386.857,167.955,49.621,159.244
C05220=1022.396,140.908,386.837,167.958,49.616,159.244
C05221=1022.401,141.157,386.816,167.961,49.610,159.243
C05222=1022.407,141.406,386.796,167.964,49.604,159.243
C05223=1022.412,141.655,386.776,167.967,49.599,159.242
C05224=1022.417,141.904,386.755,167.971,49.594,159.241
C05225=1022.423,142.153,386.734,167.973,49.588,159.241
C05226=1022.429,142.402,386.714,167.976,49.582,159.240
C05227=1022.434,142.651,386.694,167.980,49.576,159.240
C05228=1022.440,142.901,386.673,167.983,49.571,159.239
C05229=1022.445,143.150,386.652,167.986,49.565,159.238
C05230=1022.451,143.399,386.632,167.989,49.559,159.238
C05231=1022.456,143.648,386.612,167.992,49.554,159.237
C05232=1022.461,143.897,386.591,167.995,49.548,159.236
C05233=1022.467,144.147,386.571,167.998,49.542,159.236
C05234=1022.473,144.395,386.551,168.002,49.536,159.235
C05235=1022.478,144.644,386.530,168.005,49.531,159.234
C05236=1022.484,144.894,386.509,168.008,49.525,159.234
C05237=1022.489,145.143,386.489,168.011,49.520,159.233
C05238=1022.495,145.392,386.468,168.014,49.514,159.232
C05239=1022.501,145.641,386.448,168.018,49.508,159.232
C05240=1022.506,145.890,386.427,168.021,49.503,159.231
C05241=1022.511,146.139,386.406,168.024,49.497,159.231
C05242=1022.517,146.389,386.386,168.027,49.492,159.230
C05243=1022.522,146.638,386.365,168.030,49.486,159.229
C05244=1022.528,146.886,386.344,168.033,49.480,159.229
C05245=1022.533,147.136,386.323,168.036,49.475,159.228
C05246=1022.538,147.385,386.303,168.040,49.469,159.227
C05247=1022.544,147.635,386.282,168.044,49.464,159.227
C05248=1022.550,147.883,386.261,168.047,49.458,159.226
C05249=1022.556,148.132,386.240,168.050,49.453,159.226
C05250=1022.561,148.381,386.220,168.052,49.447,159.225
C05251=1022.567,148.629,386.199,168.055,49.441,159.224
C05252=1022.572,148.879,386.178,168.059,49.435,159.224
C05253=1022.578,149.128,386.157,168.062,49.430,159.223
C05254=1022.583,149.377,386.136,168.066,49.425,159.223
C05255=1022.589,149.626,386.115,168.069,49.419,159.222
C05256=1022.594,149.875,386.095,168.072,49.414,159.221
C05257=1022.600,150.124,386.073,168.075,49.408,159.221
C05258=1022.604,150.374,386.052,168.079,49.402,159.220
C05259=1022.610,150.623,386.031,168.082,49.396,159.219
C05260=1022.615,150.871,386.010,168.085,49.391,159.219
C05261=1022.621,151.121,385.989,168.088,49.386,159.218
C05262=1022.627,151.370,385.968,168.091,49.380,159.218
C05263=1022.632,151.619,385.947,168.094,49.374,159.217
C05264=1022.637,151.868,385.927,168.098,49.369,159.216
C05265=1022.643,152.117,385.905,168.101,49.363,159.216
C05266=1022.649,152.366,385.885,168.104,49.358,159.215
C05267=1022.654,152.615,385.863,168.107,49.352,159.215
C05268=1022.659,152.864,385.843,168.111,49.346,159.214
C05269=1022.666,153.113,385.821,168.114,49.341,159.213
C05270=1022.671,153.362,385.801,168.117,49.335,159.213
C05271=1022.676,153.611,385.779,168.120,49.330,159.212
C05272=1022.682,153.861,385.759,168.124,49.325,159.212
C05273=1022.687,154.109,385.737,168.128,49.319,159.211
C05274=1022.692,154.359,385.716,168.131,49.313,159.210
C05275=1022.699,154.608,385.694,168.134,49.307,159.210
C05276=1022.704,154.857,385.674,168.137,49.303,159.209
C05277=1022.709,155.105,385.653,168.140,49.297,159.209
C05278=1022.716,155.388,385.628,168.144,49.290,159.208
C05279=1022.722,155.671,385.605,168.148,49.284,159.207
C05280=1022.728,155.954,385.580,168.151,49.278,159.206
C05281=1022.734,156.237,385.557,168.155,49.272,159.206
C05282=1022.739,156.486,385.535,168.158,49.266,159.205
C05283=1022.745,156.736,385.513,168.162,49.260,159.205
C05284=1022.751,156.985,385.493,168.165,49.255,159.204
C05285=1022.756,157.233,385.471,168.168,49.249,159.203
C05286=1022.762,157.482,385.450,168.172,49.244,159.203
C05287=1022.767,157.732,385.429,168.176,49.238,159.202
C05288=1022.773,157.981,385.407,168.179,49.233,159.202
C05289=1022.779,158.229,385.386,168.182,49.227,159.201
C05290=1022.784,158.479,385.365,168.185,49.222,159.200
C05291=1022.790,158.728,385.343,168.189,49.216,159.200
C05292=1022.795,158.977,385.322,168.192,49.211,159.199
C05293=1022.801,159.226,385.300,168.195,49.205,159.199
C05294=1022.806,159.475,385.278,168.198,49.200,159.198
C05295=1022.811,159.724,385.258,168.201,49.195,159.197
C05296=1022.817,159.973,385.235,168.205,49.190,159.197
C05297=1022.821,160.222,385.213,168.209,49.184,159.196
C05298=1022.827,160.471,385.192,168.212,49.178,159.196
C05299=1022.832,160.720,385.170,168.215,49.173,159.195
C05300=1022.837,160.969,385.148,168.218,49.168,159.195
C05301=1022.843,161.217,385.127,168.222,49.163,159.194
C05302=1022.848,161.467,385.105,168.226,49.157,159.194
C05303=1022.853,161.716,385.083,168.229,49.152,159.193
C05304=1022.859,161.965,385.061,168.232,49.146,159.192
C05305=1022.864,162.214,385.039,168.235,49.141,159.192
C05306=1022.870,162.462,385.018,168.238,49.136,159.191
C05307=1022.875,162.712,384.996,168.242,49.130,159.191
C05308=1022.880,162.961,384.974,168.246,49.125,159.190
C05309=1022.886,163.210,384.952,168.249,49.119,159.190
C05310=1022.891,163.459,384.930,168.252,49.115,159.189
C05311=1022.896,163.708,384.908,168.255,49.109,159.188
C05312=1022.902,163.957,384.887,168.260,49.104,159.188
C05313=1022.907,164.205,384.865,168.263,49.098,159.187
C05314=1022.912,164.455,384.843,168.266,49.093,159.187
C05315=1022.918,164.704,384.821,168.269,49.088,159.186
C05316=1022.923,164.952,384.799,168.273,49.082,159.186
C05317=1022.928,165.201,384.777,168.276,49.077,159.185
C05318=1022.934,165.450,384.755,168.279,49.071,159.184
C05319=1022.939,165.699,384.733,168.283,49.066,159.184
C05320=1022.945,165.949,384.711,168.287,49.061,159.183
C05321=1022.950,166.197,384.690,168.290,49.056,159.183
C05322=1022.955,166.447,384.667,168.293,49.050,159.182
C05323=1022.960,166.696,384.646,168.296,49.045,159.182
C05324=1022.967,166.944,384.623,168.301,49.039,159.181
C05325=1022.972,167.193,384.601,168.304,49.034,159.181
C05326=1022.977,167.443,384.579,168.307,49.029,159.180
C05327=1022.983,167.691,384.558,168.311,49.023,159.179
C05328=1022.988,167.941,384.536,168.314,49.018,159.179
C05329=1022.993,168.189,384.514,168.317,49.013,159.178
C05330=1022.999,168.438,384.491,168.320,49.007,159.178
C05331=1023.004,168.687,384.470,168.325,49.002,159.177
C05332=1023.010,168.936,384.447,168.328,48.996,159.177
C05333=1023.016,169.185,384.426,168.331,48.991,159.176
C05334=1023.021,169.434,384.403,168.335,48.985,159.176
C05335=1023.026,169.683,384.381,168.339,48.981,159.175
C05336=1023.032,169.932,384.360,168.342,48.975,159.174
C05337=1023.037,170.181,384.337,168.346,48.969,159.174
C05338=1023.042,170.429,384.315,168.349,48.964,159.173
C05339=1023.049,170.679,384.293,168.352,48.959,159.173
C05340=1023.054,170.928,384.271,168.357,48.953,159.172
C05341=1023.059,171.177,384.249,168.360,48.948,159.172
C05342=1023.066,171.459,384.224,168.364,48.942,159.171
C05343=1023.072,171.742,384.198,168.367,48.936,159.170
C05344=1023.079,172.025,384.174,168.371,48.930,159.170
C05345=1023.085,172.307,384.148,168.376,48.924,159.169
C05346=1023.089,172.556,384.126,168.380,48.918,159.169
C05347=1023.096,172.805,384.104,168.383,48.913,159.168
C05348=1023.101,173.054,384.082,168.387,48.907,159.167
C05349=1023.106,173.303,384.060,168.390,48.902,159.167
C05350=1023.113,173.552,384.037,168.393,48.897,159.166
C05351=1023.118,173.801,384.015,168.398,48.891,159.166
C05352=1023.123,174.050,383.993,168.401,48.886,159.165
C05353=1023.129,174.298,383.971,168.404,48.881,159.165
C05354=1023.135,174.548,383.949,168.408,48.875,159.164
C05355=1023.140,174.796,383.926,168.411,48.870,159.164
C05356=1023.146,175.045,383.904,168.416,48.865,159.163
C05357=1023.152,175.294,383.881,168.419,48.859,159.162
C05358=1023.157,175.544,383.859,168.423,48.853,159.162
C05359=1023.162,175.792,383.837,168.426,48.848,159.161
C05360=1023.168,176.041,383.815,168.429,48.843,159.161
C05361=1023.174,176.291,383.793,168.434,48.838,159.160
C05362=1023.180,176.540,383.770,168.437,48.832,159.160
C05363=1023.185,176.788,383.749,168.441,48.827,159.159
C05364=1023.191,177.037,383.726,168.444,48.821,159.159
C05365=1023.196,177.287,383.703,168.448,48.816,159.158
C05366=1023.203,177.535,383.681,168.452,48.811,159.158
C05367=1023.208,177.783,383.658,168.456,48.805,159.157
C05368=1023.213,178.033,383.636,168.459,48.800,159.156
C05369=1023.219,178.282,383.613,168.463,48.794,159.156
C05370=1023.225,178.531,383.592,168.467,48.789,159.155
C05371=1023.230,178.779,383.569,168.471,48.784,159.155
C05372=1023.236,179.029,383.547,168.474,48.779,159.154
C05373=1023.242,179.277,383.525,168.477,48.773,159.154
C05374=1023.248,179.526,383.502,168.481,48.767,159.153
C05375=1023.253,179.776,383.479,168.485,48.762,159.153
C05376=1023.259,180.025,383.456,168.489,48.757,159.152
C05377=1023.265,180.273,383.435,168.492,48.752,159.151
C05378=1023.270,180.522,383.412,168.496,48.746,159.151
C05379=1023.276,180.771,383.389,168.501,48.741,159.151
C05380=1023.282,181.020,383.368,168.504,48.735,159.150
C05381=1023.288,181.269,383.345,168.508,48.730,159.149
C05382=1023.294,181.518,383.322,168.511,48.725,159.149
C05383=1023.299,181.767,383.299,168.516,48.719,159.148
C05384=1023.305,182.015,383.277,168.519,48.714,159.148
C05385=1023.311,182.264,383.255,168.523,48.708,159.147
C05386=1023.317,182.513,383.232,168.526,48.703,159.147
C05387=1023.322,182.762,383.209,168.531,48.698,159.146
C05388=1023.327,183.012,383.186,168.534,48.693,159.146
C05389=1023.333,183.261,383.163,168.537,48.688,159.145
C05390=1023.338,183.510,383.139,168.541,48.683,159.145
C05391=1023.343,183.759,383.116,168.545,48.678,159.144
C05392=1023.349,184.007,383.094,168.549,48.673,159.144
C05393=1023.354,184.256,383.070,168.553,48.668,159.143
C05394=1023.359,184.505,383.047,168.556,48.662,159.143
C05395=1023.365,184.754,383.024,168.560,48.657,159.142
C05396=1023.370,185.003,383.000,168.564,48.652,159.142
C05397=1023.376,185.251,382.977,168.568,48.647,159.141
C05398=1023.382,185.500,382.954,168.571,48.642,159.141
C05399=1023.386,185.749,382.931,168.575,48.637,159.140
C05400=1023.392,185.998,382.908,168.579,48.632,159.140
C05401=1023.398,186.247,382.885,168.582,48.627,159.139
C05402=1023.403,186.496,382.862,168.587,48.622,159.139
C05403=1023.408,186.745,382.839,168.590,48.616,159.138
C05404=1023.414,186.994,382.816,168.594,48.611,159.138
C05405=1023.419,187.243,382.792,168.598,48.606,159.137
C05406=1023.425,187.525,382.766,168.603,48.600,159.137
C05407=1023.432,187.806,382.739,168.607,48.594,159.136
C05408=1023.438,188.088,382.713,168.611,48.589,159.136
C05409=1023.445,188.371,382.687,168.615,48.583,159.135
C05410=1023.450,188.620,382.663,168.619,48.578,159.135
C05411=1023.456,188.869,382.640,168.623,48.573,159.134
C05412=1023.461,189.117,382.617,168.627,48.568,159.134
C05413=1023.466,189.366,382.594,168.631,48.563,159.133
C05414=1023.472,189.614,382.570,168.635,48.558,159.133
C05415=1023.477,189.864,382.547,168.638,48.552,159.132
C05416=1023.482,190.113,382.524,168.643,48.547,159.132
C05417=1023.488,190.361,382.501,168.646,48.542,159.131
C05418=1023.494,190.610,382.476,168.651,48.537,159.131
C05419=1023.499,190.859,382.453,168.654,48.532,159.130
C05420=1023.505,191.108,382.430,168.658,48.527,159.130
C05421=1023.511,191.358,382.407,168.662,48.521,159.129
C05422=1023.517,191.606,382.383,168.666,48.517,159.129
C05423=1023.522,191.855,382.360,168.670,48.512,159.128
C05424=1023.527,192.104,382.336,168.674,48.507,159.128
C05425=1023.533,192.352,382.313,168.678,48.502,159.127
C05426=1023.538,192.602,382.289,168.681,48.496,159.127
C05427=1023.544,192.850,382.266,168.686,48.491,159.126
C05428=1023.550,193.099,382.243,168.690,48.486,159.126
C05429=1023.555,193.348,382.219,168.694,48.481,159.125
C05430=1023.561,193.596,382.195,168.698,48.476,159.125
C05431=1023.567,193.845,382.172,168.701,48.471,159.125
C05432=1023.572,194.094,382.149,168.706,48.465,159.124
C05433=1023.578,194.343,382.125,168.710,48.460,159.124
C05434=1023.583,194.592,382.102,168.713,48.456,159.123
C05435=1023.590,194.841,382.078,168.718,48.450,159.123
C05436=1023.595,195.090,382.055,168.721,48.446,159.122
C05437=1023.601,195.338,382.030,168.726,48.440,159.122
C05438=1023.606,195.587,382.008,168.730,48.435,159.121
C05439=1023.612,195.835,381.984,168.733,48.430,159.121
C05440=1023.617,196.085,381.960,168.738,48.425,159.120
C05441=1023.624,196.334,381.936,168.742,48.420,159.120
C05442=1023.629,196.583,381.913,168.746,48.415,159.119
C05443=1023.635,196.831,381.889,168.750,48.410,159.119
C05444=1023.641,197.080,381.866,168.754,48.405,159.119
C05445=1023.646,197.329,381.842,168.758,48.400,159.118
C05446=1023.652,197.578,381.819,168.762,48.395,159.118
C05447=1023.658,197.827,381.794,168.766,48.389,159.117
C05448=1023.664,198.075,381.771,168.770,48.384,159.117
C05449=1023.669,198.324,381.748,168.774,48.379,159.116
C05450=1023.675,198.573,381.723,168.779,48.374,159.116
C05451=1023.681,198.822,381.700,168.782,48.369,159.115
C05452=1023.686,199.071,381.676,168.787,48.364,159.115
C05453=1023.692,199.319,381.652,168.791,48.359,159.114
C05454=1023.698,199.568,381.629,168.795,48.354,159.114
C05455=1023.704,199.817,381.605,168.799,48.349,159.113
C05456=1023.709,200.066,381.580,168.803,48.344,159.113
C05457=1023.715,200.314,381.557,168.807,48.339,159.113
C05458=1023.720,200.563,381.533,168.811,48.334,159.112
C05459=1023.726,200.813,381.509,168.816,48.329,159.112
C05460=1023.732,201.061,381.484,168.819,48.324,159.111
C05461=1023.738,201.309,381.461,168.824,48.319,159.111
C05462=1023.743,201.558,381.436,168.828,48.314,159.110
